(* PLC project Iec Unit Test, CODESYS CODESYS V3.5 SP16, author Toni Kucic *)
(* stored: creationDateTime 2021-05-10T20:20:27.8904239, version 0.1, modificationDateTime 2021-05-10T20:20:18.2154107, organization TK Automation *)
(* Library written in pure IEC 61131-3 Structured text that can be used for unit testing of any PLC POU. This library has arisen from the need of having a manufacturer and IDE independent unit test framework that is easily portable to other platform as the community requires. There are good unit frameworks existing for TwinCat, Codesys, B&R and many more platforms but none of them quite solve the extreme cases. *)

TYPE utTestCase : STRUCT
  id : UINT;  (* Identifier of the test *)
  desc : ARRAY[0..4] OF STRING(255);  (* Description of the test case *)
  state : utTestCaseStates;  (* State of the test *)
  msg : STRING(255);  (* Result of the test *)
END_STRUCT;
END_TYPE

(* values of utTestCaseStates: SETUP: Test case in setup mode, ready for execution; RUNNING: Test case running; PASSED: Test case passed; FAILED: Test case failed *)

{attribute 'qualified_only'}
{attribute 'strict'}
TYPE utTestCaseStates : (SETUP := 0, RUNNING := 1, PASSED := 2, FAILED := 3);
END_TYPE

TYPE utTestCaseSummary : STRUCT
  Id : UINT;  (* Id of the test object. Must be unique number *)
  Name : STRING(250);  (* Name of the test object *)
  TotalTests : UINT;  (* Total number of tests existing *)
  TestsPassed : UINT;  (* Number of tests passed *)
  TestsFailed : UINT;  (* Number of tests failed *)
  PassRate : REAL;  (* Pass rate % of the tests *)
  TestsRunning : BOOL;  (* One or more tests are running *)
  Error : utErrors := utErrors.NO_ERROR;  (* Error code if error occured *)
END_STRUCT;
END_TYPE

(* values of utErrors: NO_ERROR: No errors detected; NO_TEST_CASES_DEFINED: No test cases defined for this POU *)

{attribute 'qualified_only'}
{attribute 'strict'}
TYPE utErrors : (NO_ERROR := 0, NO_TEST_CASES_DEFINED := 100);
END_TYPE

FUNCTION assertFalse : BOOL
  VAR_INPUT
    condition : BOOL;  (* Variable to test *)
  END_VAR

            assertFalse := NOT condition;
RETURN;

          
END_FUNCTION

FUNCTION assertEqual_BOOL : BOOL
  VAR_INPUT
    act : BOOL;  (* Variable to test *)
    xp : BOOL;  (* Variable to test against *)
  END_VAR

            assertEqual_BOOL := act = xp;
RETURN;

          
END_FUNCTION

FUNCTION assertEqual_BYTE : BOOL
  VAR_INPUT
    act : BYTE;  (* Variable to test *)
    xp : BYTE;  (* Variable to test against *)
  END_VAR

            assertEqual_BYTE := act = xp;
RETURN;

          
END_FUNCTION

FUNCTION assertEqual_WORD : BOOL
  VAR_INPUT
    act : WORD;  (* Variable to test *)
    xp : WORD;  (* Variable to test against *)
  END_VAR

            assertEqual_WORD := act = xp;
RETURN;

          
END_FUNCTION

FUNCTION assertEqual_DWORD : BOOL
  VAR_INPUT
    act : DWORD;  (* Variable to test *)
    xp : DWORD;  (* Variable to test against *)
  END_VAR

            assertEqual_DWORD := act = xp;
RETURN;

          
END_FUNCTION

FUNCTION assertEqual_LWORD : BOOL
  VAR_INPUT
    act : LWORD;  (* Variable to test *)
    xp : LWORD;  (* Variable to test against *)
  END_VAR

            assertEqual_LWORD := act = xp;
RETURN;

          
END_FUNCTION

FUNCTION assertEqual_SINT : BOOL
  VAR_INPUT
    act : SINT;  (* Variable to test *)
    xp : SINT;  (* Variable to test against *)
  END_VAR

            assertEqual_SINT := act = xp;
RETURN;

          
END_FUNCTION

FUNCTION assertEqual_USINT : BOOL
  VAR_INPUT
    act : USINT;  (* Variable to test *)
    xp : USINT;  (* Variable to test against *)
  END_VAR

            assertEqual_USINT := act = xp;
RETURN;

          
END_FUNCTION

FUNCTION assertEqual_INT : BOOL
  VAR_INPUT
    act : INT;  (* Variable to test *)
    xp : INT;  (* Variable to test against *)
  END_VAR

            assertEqual_INT := act = xp;
RETURN;

          
END_FUNCTION

FUNCTION assertEqual_UINT : BOOL
  VAR_INPUT
    act : UINT;  (* Variable to test *)
    xp : UINT;  (* Variable to test against *)
  END_VAR

            assertEqual_UINT := act = xp;
RETURN;

          
END_FUNCTION

FUNCTION assertEqual_DINT : BOOL
  VAR_INPUT
    act : DINT;  (* Variable to test *)
    xp : DINT;  (* Variable to test against *)
  END_VAR

            assertEqual_DINT := act = xp;
RETURN;

          
END_FUNCTION

FUNCTION assertEqual_UDINT : BOOL
  VAR_INPUT
    act : UDINT;  (* Variable to test *)
    xp : UDINT;  (* Variable to test against *)
  END_VAR

            assertEqual_UDINT := act = xp;
RETURN;

          
END_FUNCTION

FUNCTION assertEqual_LINT : BOOL
  VAR_INPUT
    act : LINT;  (* Variable to test *)
    xp : LINT;  (* Variable to test against *)
  END_VAR

            assertEqual_LINT := act = xp;
RETURN;

          
END_FUNCTION

FUNCTION assertEqual_ULINT : BOOL
  VAR_INPUT
    act : ULINT;  (* Variable to test *)
    xp : ULINT;  (* Variable to test against *)
  END_VAR

            assertEqual_ULINT := act = xp;
RETURN;

          
END_FUNCTION

FUNCTION assertEqual_REAL : BOOL
  VAR_INPUT
    act : REAL;  (* Variable to test *)
    xp : REAL;  (* Variable to test against *)
  END_VAR

            assertEqual_REAL := act = xp;
RETURN;

          
END_FUNCTION

FUNCTION assertEqual_LREAL : BOOL
  VAR_INPUT
    act : LREAL;  (* Variable to test *)
    xp : LREAL;  (* Variable to test against *)
  END_VAR

            assertEqual_LREAL := act = xp;
RETURN;

          
END_FUNCTION

FUNCTION assertEqual_STRING : BOOL
  VAR_INPUT
    act : STRING;  (* Variable to test *)
    xp : STRING;  (* Variable to test against *)
  END_VAR

            assertEqual_STRING := act = xp;
RETURN;

          
END_FUNCTION

FUNCTION assertEqual_WSTRING : BOOL
  VAR_INPUT
    act : WSTRING;  (* Variable to test *)
    xp : WSTRING;  (* Variable to test against *)
  END_VAR

            assertEqual_WSTRING := act = xp;
RETURN;

          
END_FUNCTION

FUNCTION assertEqual_TIME : BOOL
  VAR_INPUT
    act : TIME;  (* Variable to test *)
    xp : TIME;  (* Variable to test against *)
  END_VAR

            assertEqual_TIME := act = xp;
RETURN;

          
END_FUNCTION

FUNCTION assertEqual_LTIME : BOOL
  VAR_INPUT
    act : LTIME;  (* Variable to test *)
    xp : LTIME;  (* Variable to test against *)
  END_VAR

            assertEqual_LTIME := act = xp;
RETURN;

          
END_FUNCTION

FUNCTION assertEqual_DATE : BOOL
  VAR_INPUT
    act : DATE;  (* Variable to test *)
    xp : DATE;  (* Variable to test against *)
  END_VAR

            assertEqual_DATE := act = xp;
RETURN;

          
END_FUNCTION

FUNCTION assertEqual_LDATE : BOOL
  VAR_INPUT
    act : LDATE;  (* Variable to test *)
    xp : LDATE;  (* Variable to test against *)
  END_VAR

            assertEqual_LDATE := act = xp;
RETURN;

          
END_FUNCTION

FUNCTION assertEqual_DATE_AND_TIME : BOOL
  VAR_INPUT
    act : DT;  (* Variable to test *)
    xp : DT;  (* Variable to test against *)
  END_VAR

            assertEqual_DATE_AND_TIME := act = xp;
RETURN;

          
END_FUNCTION

FUNCTION assertEqual_LDATE_AND_TIME : BOOL
  VAR_INPUT
    act : LDATE_AND_TIME;  (* Variable to test *)
    xp : LDATE_AND_TIME;  (* Variable to test against *)
  END_VAR

            assertEqual_LDATE_AND_TIME := act = xp;
RETURN;

          
END_FUNCTION

FUNCTION assertEqual_TIME_OF_DAY : BOOL
  VAR_INPUT
    act : TOD;  (* Variable to test *)
    xp : TOD;  (* Variable to test against *)
  END_VAR

            assertEqual_TIME_OF_DAY := act = xp;
RETURN;

          
END_FUNCTION

FUNCTION assertEqual_LTIME_OF_DAY : BOOL
  VAR_INPUT
    act : LTIME_OF_DAY;  (* Variable to test *)
    xp : LTIME_OF_DAY;  (* Variable to test against *)
  END_VAR

            assertEqual_LTIME_OF_DAY := act = xp;
RETURN;

          
END_FUNCTION

FUNCTION assertNotEqual_BOOL : BOOL
  VAR_INPUT
    act : BOOL;  (* Variable to test *)
    xp : BOOL;  (* Variable to test against *)
  END_VAR

            assertNotEqual_BOOL := act <> xp;
RETURN;

          
END_FUNCTION

FUNCTION assertNotEqual_BYTE : BOOL
  VAR_INPUT
    act : BYTE;  (* Variable to test *)
    xp : BYTE;  (* Variable to test against *)
  END_VAR

            assertNotEqual_BYTE := act <> xp;
RETURN;

          
END_FUNCTION

FUNCTION assertNotEqual_WORD : BOOL
  VAR_INPUT
    act : WORD;  (* Variable to test *)
    xp : WORD;  (* Variable to test against *)
  END_VAR

            assertNotEqual_WORD := act <> xp;
RETURN;

          
END_FUNCTION

FUNCTION assertNotEqual_DWORD : BOOL
  VAR_INPUT
    act : DWORD;  (* Variable to test *)
    xp : DWORD;  (* Variable to test against *)
  END_VAR

            assertNotEqual_DWORD := act <> xp;
RETURN;

          
END_FUNCTION

FUNCTION assertNotEqual_LWORD : BOOL
  VAR_INPUT
    act : LWORD;  (* Variable to test *)
    xp : LWORD;  (* Variable to test against *)
  END_VAR

            assertNotEqual_LWORD := act <> xp;
RETURN;

          
END_FUNCTION

FUNCTION assertNotEqual_SINT : BOOL
  VAR_INPUT
    act : SINT;  (* Variable to test *)
    xp : SINT;  (* Variable to test against *)
  END_VAR

            assertNotEqual_SINT := act <> xp;
RETURN;

          
END_FUNCTION

FUNCTION assertNotEqual_USINT : BOOL
  VAR_INPUT
    act : USINT;  (* Variable to test *)
    xp : USINT;  (* Variable to test against *)
  END_VAR

            assertNotEqual_USINT := act <> xp;
RETURN;

          
END_FUNCTION

FUNCTION assertNotEqual_INT : BOOL
  VAR_INPUT
    act : INT;  (* Variable to test *)
    xp : INT;  (* Variable to test against *)
  END_VAR

            assertNotEqual_INT := act <> xp;
RETURN;

          
END_FUNCTION

FUNCTION assertNotEqual_UINT : BOOL
  VAR_INPUT
    act : UINT;  (* Variable to test *)
    xp : UINT;  (* Variable to test against *)
  END_VAR

            assertNotEqual_UINT := act <> xp;
RETURN;

          
END_FUNCTION

FUNCTION assertNotEqual_DINT : BOOL
  VAR_INPUT
    act : DINT;  (* Variable to test *)
    xp : DINT;  (* Variable to test against *)
  END_VAR

            assertNotEqual_DINT := act <> xp;
RETURN;

          
END_FUNCTION

FUNCTION assertNotEqual_UDINT : BOOL
  VAR_INPUT
    act : UDINT;  (* Variable to test *)
    xp : UDINT;  (* Variable to test against *)
  END_VAR

            assertNotEqual_UDINT := act <> xp;
RETURN;

          
END_FUNCTION

FUNCTION assertNotEqual_LINT : BOOL
  VAR_INPUT
    act : LINT;  (* Variable to test *)
    xp : LINT;  (* Variable to test against *)
  END_VAR

            assertNotEqual_LINT := act <> xp;
RETURN;

          
END_FUNCTION

FUNCTION assertNotEqual_ULINT : BOOL
  VAR_INPUT
    act : ULINT;  (* Variable to test *)
    xp : ULINT;  (* Variable to test against *)
  END_VAR

            assertNotEqual_ULINT := act <> xp;
RETURN;

          
END_FUNCTION

FUNCTION assertNotEqual_REAL : BOOL
  VAR_INPUT
    act : REAL;  (* Variable to test *)
    xp : REAL;  (* Variable to test against *)
  END_VAR

            assertNotEqual_REAL := act <> xp;
RETURN;

          
END_FUNCTION

FUNCTION assertNotEqual_LREAL : BOOL
  VAR_INPUT
    act : LREAL;  (* Variable to test *)
    xp : LREAL;  (* Variable to test against *)
  END_VAR

            assertNotEqual_LREAL := act <> xp;
RETURN;

          
END_FUNCTION

FUNCTION assertNotEqual_STRING : BOOL
  VAR_INPUT
    act : STRING;  (* Variable to test *)
    xp : STRING;  (* Variable to test against *)
  END_VAR

            assertNotEqual_STRING := act <> xp;
RETURN;

          
END_FUNCTION

FUNCTION assertNotEqual_WSTRING : BOOL
  VAR_INPUT
    act : WSTRING;  (* Variable to test *)
    xp : WSTRING;  (* Variable to test against *)
  END_VAR

            assertNotEqual_WSTRING := act <> xp;
RETURN;

          
END_FUNCTION

FUNCTION assertNotEqual_TIME : BOOL
  VAR_INPUT
    act : TIME;  (* Variable to test *)
    xp : TIME;  (* Variable to test against *)
  END_VAR

            assertNotEqual_TIME := act <> xp;
RETURN;

          
END_FUNCTION

FUNCTION assertNotEqual_LTIME : BOOL
  VAR_INPUT
    act : LTIME;  (* Variable to test *)
    xp : LTIME;  (* Variable to test against *)
  END_VAR

            assertNotEqual_LTIME := act <> xp;
RETURN;

          
END_FUNCTION

FUNCTION assertNotEqual_DATE : BOOL
  VAR_INPUT
    act : DATE;  (* Variable to test *)
    xp : DATE;  (* Variable to test against *)
  END_VAR

            assertNotEqual_DATE := act <> xp;
RETURN;

          
END_FUNCTION

FUNCTION assertNotEqual_LDATE : BOOL
  VAR_INPUT
    act : LDATE;  (* Variable to test *)
    xp : LDATE;  (* Variable to test against *)
  END_VAR

            assertNotEqual_LDATE := act <> xp;
RETURN;

          
END_FUNCTION

FUNCTION assertNotEqual_DATE_AND_TIME : BOOL
  VAR_INPUT
    act : DT;  (* Variable to test *)
    xp : DT;  (* Variable to test against *)
  END_VAR

            assertNotEqual_DATE_AND_TIME := act <> xp;
RETURN;

          
END_FUNCTION

FUNCTION assertNotEqual_LDATE_AND_TIME : BOOL
  VAR_INPUT
    act : LDATE_AND_TIME;  (* Variable to test *)
    xp : LDATE_AND_TIME;  (* Variable to test against *)
  END_VAR

            assertNotEqual_LDATE_AND_TIME := act <> xp;
RETURN;

          
END_FUNCTION

FUNCTION assertNotEqual_TIME_OF_DAY : BOOL
  VAR_INPUT
    act : TOD;  (* Variable to test *)
    xp : TOD;  (* Variable to test against *)
  END_VAR

            assertNotEqual_TIME_OF_DAY := act <> xp;
RETURN;

          
END_FUNCTION

FUNCTION assertNotEqual_LTIME_OF_DAY : BOOL
  VAR_INPUT
    act : LTIME_OF_DAY;  (* Variable to test *)
    xp : LTIME_OF_DAY;  (* Variable to test against *)
  END_VAR

            assertNotEqual_LTIME_OF_DAY := act <> xp;
RETURN;

          
END_FUNCTION

FUNCTION assertGreater_BYTE : BOOL
  VAR_INPUT
    act : BYTE;  (* Variable to test *)
    xp : BYTE;  (* Variable to test against *)
  END_VAR

            assertGreater_BYTE := act > xp;
RETURN;

          
END_FUNCTION

FUNCTION assertGreater_WORD : BOOL
  VAR_INPUT
    act : WORD;  (* Variable to test *)
    xp : WORD;  (* Variable to test against *)
  END_VAR

            assertGreater_WORD := act > xp;
RETURN;

          
END_FUNCTION

FUNCTION assertGreater_DWORD : BOOL
  VAR_INPUT
    act : DWORD;  (* Variable to test *)
    xp : DWORD;  (* Variable to test against *)
  END_VAR

            assertGreater_DWORD := act > xp;
RETURN;

          
END_FUNCTION

FUNCTION assertGreater_LWORD : BOOL
  VAR_INPUT
    act : LWORD;  (* Variable to test *)
    xp : LWORD;  (* Variable to test against *)
  END_VAR

            assertGreater_LWORD := act > xp;
RETURN;

          
END_FUNCTION

FUNCTION assertGreater_SINT : BOOL
  VAR_INPUT
    act : SINT;  (* Variable to test *)
    xp : SINT;  (* Variable to test against *)
  END_VAR

            assertGreater_SINT := act > xp;
RETURN;

          
END_FUNCTION

FUNCTION assertGreater_USINT : BOOL
  VAR_INPUT
    act : USINT;  (* Variable to test *)
    xp : USINT;  (* Variable to test against *)
  END_VAR

            assertGreater_USINT := act > xp;
RETURN;

          
END_FUNCTION

FUNCTION assertGreater_INT : BOOL
  VAR_INPUT
    act : INT;  (* Variable to test *)
    xp : INT;  (* Variable to test against *)
  END_VAR

            assertGreater_INT := act > xp;
RETURN;

          
END_FUNCTION

FUNCTION assertGreater_UINT : BOOL
  VAR_INPUT
    act : UINT;  (* Variable to test *)
    xp : UINT;  (* Variable to test against *)
  END_VAR

            assertGreater_UINT := act > xp;
RETURN;

          
END_FUNCTION

FUNCTION assertGreater_DINT : BOOL
  VAR_INPUT
    act : DINT;  (* Variable to test *)
    xp : DINT;  (* Variable to test against *)
  END_VAR

            assertGreater_DINT := act > xp;
RETURN;

          
END_FUNCTION

FUNCTION assertGreater_UDINT : BOOL
  VAR_INPUT
    act : UDINT;  (* Variable to test *)
    xp : UDINT;  (* Variable to test against *)
  END_VAR

            assertGreater_UDINT := act > xp;
RETURN;

          
END_FUNCTION

FUNCTION assertGreater_LINT : BOOL
  VAR_INPUT
    act : LINT;  (* Variable to test *)
    xp : LINT;  (* Variable to test against *)
  END_VAR

            assertGreater_LINT := act > xp;
RETURN;

          
END_FUNCTION

FUNCTION assertGreater_ULINT : BOOL
  VAR_INPUT
    act : ULINT;  (* Variable to test *)
    xp : ULINT;  (* Variable to test against *)
  END_VAR

            assertGreater_ULINT := act > xp;
RETURN;

          
END_FUNCTION

FUNCTION assertGreater_REAL : BOOL
  VAR_INPUT
    act : REAL;  (* Variable to test *)
    xp : REAL;  (* Variable to test against *)
  END_VAR

            assertGreater_REAL := act > xp;
RETURN;

          
END_FUNCTION

FUNCTION assertGreater_LREAL : BOOL
  VAR_INPUT
    act : LREAL;  (* Variable to test *)
    xp : LREAL;  (* Variable to test against *)
  END_VAR

            assertGreater_LREAL := act > xp;
RETURN;

          
END_FUNCTION

FUNCTION assertGreater_TIME : BOOL
  VAR_INPUT
    act : TIME;  (* Variable to test *)
    xp : TIME;  (* Variable to test against *)
  END_VAR

            assertGreater_TIME := act > xp;
RETURN;

          
END_FUNCTION

FUNCTION assertGreater_LTIME : BOOL
  VAR_INPUT
    act : LTIME;  (* Variable to test *)
    xp : LTIME;  (* Variable to test against *)
  END_VAR

            assertGreater_LTIME := act > xp;
RETURN;

          
END_FUNCTION

FUNCTION assertGreater_DATE : BOOL
  VAR_INPUT
    act : DATE;  (* Variable to test *)
    xp : DATE;  (* Variable to test against *)
  END_VAR

            assertGreater_DATE := act > xp;
RETURN;

          
END_FUNCTION

FUNCTION assertGreater_LDATE : BOOL
  VAR_INPUT
    act : LDATE;  (* Variable to test *)
    xp : LDATE;  (* Variable to test against *)
  END_VAR

            assertGreater_LDATE := act > xp;
RETURN;

          
END_FUNCTION

FUNCTION assertGreater_DATE_AND_TIME : BOOL
  VAR_INPUT
    act : DT;  (* Variable to test *)
    xp : DT;  (* Variable to test against *)
  END_VAR

            assertGreater_DATE_AND_TIME := act > xp;
RETURN;

          
END_FUNCTION

FUNCTION assertGreater_LDATE_AND_TIME : BOOL
  VAR_INPUT
    act : LDATE_AND_TIME;  (* Variable to test *)
    xp : LDATE_AND_TIME;  (* Variable to test against *)
  END_VAR

            assertGreater_LDATE_AND_TIME := act > xp;
RETURN;

          
END_FUNCTION

FUNCTION assertGreater_TIME_OF_DAY : BOOL
  VAR_INPUT
    act : TOD;  (* Variable to test *)
    xp : TOD;  (* Variable to test against *)
  END_VAR

            assertGreater_TIME_OF_DAY := act > xp;
RETURN;

          
END_FUNCTION

FUNCTION assertGreater_LTIME_OF_DAY : BOOL
  VAR_INPUT
    act : LTIME_OF_DAY;  (* Variable to test *)
    xp : LTIME_OF_DAY;  (* Variable to test against *)
  END_VAR

            assertGreater_LTIME_OF_DAY := act > xp;
RETURN;

          
END_FUNCTION

FUNCTION assertGreaterEqual_BYTE : BOOL
  VAR_INPUT
    act : BYTE;  (* Variable to test *)
    xp : BYTE;  (* Variable to test against *)
  END_VAR

            assertGreaterEqual_BYTE := act >= xp;
RETURN;

          
END_FUNCTION

FUNCTION assertGreaterEqual_WORD : BOOL
  VAR_INPUT
    act : WORD;  (* Variable to test *)
    xp : WORD;  (* Variable to test against *)
  END_VAR

            assertGreaterEqual_WORD := act >= xp;
RETURN;

          
END_FUNCTION

FUNCTION assertGreaterEqual_DWORD : BOOL
  VAR_INPUT
    act : DWORD;  (* Variable to test *)
    xp : DWORD;  (* Variable to test against *)
  END_VAR

            assertGreaterEqual_DWORD := act >= xp;
RETURN;

          
END_FUNCTION

FUNCTION assertGreaterEqual_LWORD : BOOL
  VAR_INPUT
    act : LWORD;  (* Variable to test *)
    xp : LWORD;  (* Variable to test against *)
  END_VAR

            assertGreaterEqual_LWORD := act >= xp;
RETURN;

          
END_FUNCTION

FUNCTION assertGreaterEqual_SINT : BOOL
  VAR_INPUT
    act : SINT;  (* Variable to test *)
    xp : SINT;  (* Variable to test against *)
  END_VAR

            assertGreaterEqual_SINT := act >= xp;
RETURN;

          
END_FUNCTION

FUNCTION assertGreaterEqual_USINT : BOOL
  VAR_INPUT
    act : USINT;  (* Variable to test *)
    xp : USINT;  (* Variable to test against *)
  END_VAR

            assertGreaterEqual_USINT := act >= xp;
RETURN;

          
END_FUNCTION

FUNCTION assertGreaterEqual_INT : BOOL
  VAR_INPUT
    act : INT;  (* Variable to test *)
    xp : INT;  (* Variable to test against *)
  END_VAR

            assertGreaterEqual_INT := act >= xp;
RETURN;

          
END_FUNCTION

FUNCTION assertGreaterEqual_UINT : BOOL
  VAR_INPUT
    act : UINT;  (* Variable to test *)
    xp : UINT;  (* Variable to test against *)
  END_VAR

            assertGreaterEqual_UINT := act >= xp;
RETURN;

          
END_FUNCTION

FUNCTION assertGreaterEqual_DINT : BOOL
  VAR_INPUT
    act : DINT;  (* Variable to test *)
    xp : DINT;  (* Variable to test against *)
  END_VAR

            assertGreaterEqual_DINT := act >= xp;
RETURN;

          
END_FUNCTION

FUNCTION assertGreaterEqual_UDINT : BOOL
  VAR_INPUT
    act : UDINT;  (* Variable to test *)
    xp : UDINT;  (* Variable to test against *)
  END_VAR

            assertGreaterEqual_UDINT := act >= xp;
RETURN;

          
END_FUNCTION

FUNCTION assertGreaterEqual_LINT : BOOL
  VAR_INPUT
    act : LINT;  (* Variable to test *)
    xp : LINT;  (* Variable to test against *)
  END_VAR

            assertGreaterEqual_LINT := act >= xp;
RETURN;

          
END_FUNCTION

FUNCTION assertGreaterEqual_ULINT : BOOL
  VAR_INPUT
    act : ULINT;  (* Variable to test *)
    xp : ULINT;  (* Variable to test against *)
  END_VAR

            assertGreaterEqual_ULINT := act >= xp;
RETURN;

          
END_FUNCTION

FUNCTION assertGreaterEqual_REAL : BOOL
  VAR_INPUT
    act : REAL;  (* Variable to test *)
    xp : REAL;  (* Variable to test against *)
  END_VAR

            assertGreaterEqual_REAL := act >= xp;
RETURN;

          
END_FUNCTION

FUNCTION assertGreaterEqual_LREAL : BOOL
  VAR_INPUT
    act : LREAL;  (* Variable to test *)
    xp : LREAL;  (* Variable to test against *)
  END_VAR

            assertGreaterEqual_LREAL := act >= xp;
RETURN;

          
END_FUNCTION

FUNCTION assertGreaterEqual_TIME : BOOL
  VAR_INPUT
    act : TIME;  (* Variable to test *)
    xp : TIME;  (* Variable to test against *)
  END_VAR

            assertGreaterEqual_TIME := act >= xp;
RETURN;

          
END_FUNCTION

FUNCTION assertGreaterEqual_LTIME : BOOL
  VAR_INPUT
    act : LTIME;  (* Variable to test *)
    xp : LTIME;  (* Variable to test against *)
  END_VAR

            assertGreaterEqual_LTIME := act >= xp;
RETURN;

          
END_FUNCTION

FUNCTION assertGreaterEqual_DATE : BOOL
  VAR_INPUT
    act : DATE;  (* Variable to test *)
    xp : DATE;  (* Variable to test against *)
  END_VAR

            assertGreaterEqual_DATE := act >= xp;
RETURN;

          
END_FUNCTION

FUNCTION assertGreaterEqual_LDATE : BOOL
  VAR_INPUT
    act : LDATE;  (* Variable to test *)
    xp : LDATE;  (* Variable to test against *)
  END_VAR

            assertGreaterEqual_LDATE := act >= xp;
RETURN;

          
END_FUNCTION

FUNCTION assertGreaterEqual_DATE_AND_TIME : BOOL
  VAR_INPUT
    act : DT;  (* Variable to test *)
    xp : DT;  (* Variable to test against *)
  END_VAR

            assertGreaterEqual_DATE_AND_TIME := act >= xp;
RETURN;

          
END_FUNCTION

FUNCTION assertGreaterEqual_LDATE_AND_TIME : BOOL
  VAR_INPUT
    act : LDATE_AND_TIME;  (* Variable to test *)
    xp : LDATE_AND_TIME;  (* Variable to test against *)
  END_VAR

            assertGreaterEqual_LDATE_AND_TIME := act >= xp;
RETURN;

          
END_FUNCTION

FUNCTION assertGreaterEqual_TIME_OF_DAY : BOOL
  VAR_INPUT
    act : TOD;  (* Variable to test *)
    xp : TOD;  (* Variable to test against *)
  END_VAR

            assertGreaterEqual_TIME_OF_DAY := act >= xp;
RETURN;

          
END_FUNCTION

FUNCTION assertGreaterEqual_LTIME_OF_DAY : BOOL
  VAR_INPUT
    act : LTIME_OF_DAY;  (* Variable to test *)
    xp : LTIME_OF_DAY;  (* Variable to test against *)
  END_VAR

            assertGreaterEqual_LTIME_OF_DAY := act >= xp;
RETURN;

          
END_FUNCTION

FUNCTION assertLess_BYTE : BOOL
  VAR_INPUT
    act : BYTE;  (* Variable to test *)
    xp : BYTE;  (* Variable to test against *)
  END_VAR

            assertLess_BYTE := act < xp;
RETURN;

          
END_FUNCTION

FUNCTION assertLess_WORD : BOOL
  VAR_INPUT
    act : WORD;  (* Variable to test *)
    xp : WORD;  (* Variable to test against *)
  END_VAR

            assertLess_WORD := act < xp;
RETURN;

          
END_FUNCTION

FUNCTION assertLess_DWORD : BOOL
  VAR_INPUT
    act : DWORD;  (* Variable to test *)
    xp : DWORD;  (* Variable to test against *)
  END_VAR

            assertLess_DWORD := act < xp;
RETURN;

          
END_FUNCTION

FUNCTION assertLess_LWORD : BOOL
  VAR_INPUT
    act : LWORD;  (* Variable to test *)
    xp : LWORD;  (* Variable to test against *)
  END_VAR

            assertLess_LWORD := act < xp;
RETURN;

          
END_FUNCTION

FUNCTION assertLess_SINT : BOOL
  VAR_INPUT
    act : SINT;  (* Variable to test *)
    xp : SINT;  (* Variable to test against *)
  END_VAR

            assertLess_SINT := act < xp;
RETURN;

          
END_FUNCTION

FUNCTION assertLess_USINT : BOOL
  VAR_INPUT
    act : USINT;  (* Variable to test *)
    xp : USINT;  (* Variable to test against *)
  END_VAR

            assertLess_USINT := act < xp;
RETURN;

          
END_FUNCTION

FUNCTION assertLess_INT : BOOL
  VAR_INPUT
    act : INT;  (* Variable to test *)
    xp : INT;  (* Variable to test against *)
  END_VAR

            assertLess_INT := act < xp;
RETURN;

          
END_FUNCTION

FUNCTION assertLess_UINT : BOOL
  VAR_INPUT
    act : UINT;  (* Variable to test *)
    xp : UINT;  (* Variable to test against *)
  END_VAR

            assertLess_UINT := act < xp;
RETURN;

          
END_FUNCTION

FUNCTION assertLess_DINT : BOOL
  VAR_INPUT
    act : DINT;  (* Variable to test *)
    xp : DINT;  (* Variable to test against *)
  END_VAR

            assertLess_DINT := act < xp;
RETURN;

          
END_FUNCTION

FUNCTION assertLess_UDINT : BOOL
  VAR_INPUT
    act : UDINT;  (* Variable to test *)
    xp : UDINT;  (* Variable to test against *)
  END_VAR

            assertLess_UDINT := act < xp;
RETURN;

          
END_FUNCTION

FUNCTION assertLess_LINT : BOOL
  VAR_INPUT
    act : LINT;  (* Variable to test *)
    xp : LINT;  (* Variable to test against *)
  END_VAR

            assertLess_LINT := act < xp;
RETURN;

          
END_FUNCTION

FUNCTION assertLess_ULINT : BOOL
  VAR_INPUT
    act : ULINT;  (* Variable to test *)
    xp : ULINT;  (* Variable to test against *)
  END_VAR

            assertLess_ULINT := act < xp;
RETURN;

          
END_FUNCTION

FUNCTION assertLess_REAL : BOOL
  VAR_INPUT
    act : REAL;  (* Variable to test *)
    xp : REAL;  (* Variable to test against *)
  END_VAR

            assertLess_REAL := act < xp;
RETURN;

          
END_FUNCTION

FUNCTION assertLess_LREAL : BOOL
  VAR_INPUT
    act : LREAL;  (* Variable to test *)
    xp : LREAL;  (* Variable to test against *)
  END_VAR

            assertLess_LREAL := act < xp;
RETURN;

          
END_FUNCTION

FUNCTION assertLess_TIME : BOOL
  VAR_INPUT
    act : TIME;  (* Variable to test *)
    xp : TIME;  (* Variable to test against *)
  END_VAR

            assertLess_TIME := act < xp;
RETURN;

          
END_FUNCTION

FUNCTION assertLess_LTIME : BOOL
  VAR_INPUT
    act : LTIME;  (* Variable to test *)
    xp : LTIME;  (* Variable to test against *)
  END_VAR

            assertLess_LTIME := act < xp;
RETURN;

          
END_FUNCTION

FUNCTION assertLess_DATE : BOOL
  VAR_INPUT
    act : DATE;  (* Variable to test *)
    xp : DATE;  (* Variable to test against *)
  END_VAR

            assertLess_DATE := act < xp;
RETURN;

          
END_FUNCTION

FUNCTION assertLess_LDATE : BOOL
  VAR_INPUT
    act : LDATE;  (* Variable to test *)
    xp : LDATE;  (* Variable to test against *)
  END_VAR

            assertLess_LDATE := act < xp;
RETURN;

          
END_FUNCTION

FUNCTION assertLess_DATE_AND_TIME : BOOL
  VAR_INPUT
    act : DT;  (* Variable to test *)
    xp : DT;  (* Variable to test against *)
  END_VAR

            assertLess_DATE_AND_TIME := act < xp;
RETURN;

          
END_FUNCTION

FUNCTION assertLess_LDATE_AND_TIME : BOOL
  VAR_INPUT
    act : LDATE_AND_TIME;  (* Variable to test *)
    xp : LDATE_AND_TIME;  (* Variable to test against *)
  END_VAR

            assertLess_LDATE_AND_TIME := act < xp;
RETURN;

          
END_FUNCTION

FUNCTION assertLess_TIME_OF_DAY : BOOL
  VAR_INPUT
    act : TOD;  (* Variable to test *)
    xp : TOD;  (* Variable to test against *)
  END_VAR

            assertLess_TIME_OF_DAY := act < xp;
RETURN;

          
END_FUNCTION

FUNCTION assertLess_LTIME_OF_DAY : BOOL
  VAR_INPUT
    act : LTIME_OF_DAY;  (* Variable to test *)
    xp : LTIME_OF_DAY;  (* Variable to test against *)
  END_VAR

            assertLess_LTIME_OF_DAY := act < xp;
RETURN;

          
END_FUNCTION

FUNCTION assertLessEqual_BYTE : BOOL
  VAR_INPUT
    act : BYTE;  (* Variable to test *)
    xp : BYTE;  (* Variable to test against *)
  END_VAR

            assertLessEqual_BYTE := act <= xp;
RETURN;

          
END_FUNCTION

FUNCTION assertLessEqual_WORD : BOOL
  VAR_INPUT
    act : WORD;  (* Variable to test *)
    xp : WORD;  (* Variable to test against *)
  END_VAR

            assertLessEqual_WORD := act <= xp;
RETURN;

          
END_FUNCTION

FUNCTION assertLessEqual_DWORD : BOOL
  VAR_INPUT
    act : DWORD;  (* Variable to test *)
    xp : DWORD;  (* Variable to test against *)
  END_VAR

            assertLessEqual_DWORD := act <= xp;
RETURN;

          
END_FUNCTION

FUNCTION assertLessEqual_LWORD : BOOL
  VAR_INPUT
    act : LWORD;  (* Variable to test *)
    xp : LWORD;  (* Variable to test against *)
  END_VAR

            assertLessEqual_LWORD := act <= xp;
RETURN;

          
END_FUNCTION

FUNCTION assertLessEqual_SINT : BOOL
  VAR_INPUT
    act : SINT;  (* Variable to test *)
    xp : SINT;  (* Variable to test against *)
  END_VAR

            assertLessEqual_SINT := act <= xp;
RETURN;

          
END_FUNCTION

FUNCTION assertLessEqual_USINT : BOOL
  VAR_INPUT
    act : USINT;  (* Variable to test *)
    xp : USINT;  (* Variable to test against *)
  END_VAR

            assertLessEqual_USINT := act <= xp;
RETURN;

          
END_FUNCTION

FUNCTION assertLessEqual_INT : BOOL
  VAR_INPUT
    act : INT;  (* Variable to test *)
    xp : INT;  (* Variable to test against *)
  END_VAR

            assertLessEqual_INT := act <= xp;
RETURN;

          
END_FUNCTION

FUNCTION assertLessEqual_UINT : BOOL
  VAR_INPUT
    act : UINT;  (* Variable to test *)
    xp : UINT;  (* Variable to test against *)
  END_VAR

            assertLessEqual_UINT := act <= xp;
RETURN;

          
END_FUNCTION

FUNCTION assertLessEqual_DINT : BOOL
  VAR_INPUT
    act : DINT;  (* Variable to test *)
    xp : DINT;  (* Variable to test against *)
  END_VAR

            assertLessEqual_DINT := act <= xp;
RETURN;

          
END_FUNCTION

FUNCTION assertLessEqual_UDINT : BOOL
  VAR_INPUT
    act : UDINT;  (* Variable to test *)
    xp : UDINT;  (* Variable to test against *)
  END_VAR

            assertLessEqual_UDINT := act <= xp;
RETURN;

          
END_FUNCTION

FUNCTION assertLessEqual_LINT : BOOL
  VAR_INPUT
    act : LINT;  (* Variable to test *)
    xp : LINT;  (* Variable to test against *)
  END_VAR

            assertLessEqual_LINT := act <= xp;
RETURN;

          
END_FUNCTION

FUNCTION assertLessEqual_ULINT : BOOL
  VAR_INPUT
    act : ULINT;  (* Variable to test *)
    xp : ULINT;  (* Variable to test against *)
  END_VAR

            assertLessEqual_ULINT := act <= xp;
RETURN;

          
END_FUNCTION

FUNCTION assertLessEqual_REAL : BOOL
  VAR_INPUT
    act : REAL;  (* Variable to test *)
    xp : REAL;  (* Variable to test against *)
  END_VAR

            assertLessEqual_REAL := act <= xp;
RETURN;

          
END_FUNCTION

FUNCTION assertLessEqual_LREAL : BOOL
  VAR_INPUT
    act : LREAL;  (* Variable to test *)
    xp : LREAL;  (* Variable to test against *)
  END_VAR

            assertLessEqual_LREAL := act <= xp;
RETURN;

          
END_FUNCTION

FUNCTION assertLessEqual_TIME : BOOL
  VAR_INPUT
    act : TIME;  (* Variable to test *)
    xp : TIME;  (* Variable to test against *)
  END_VAR

            assertLessEqual_TIME := act <= xp;
RETURN;

          
END_FUNCTION

FUNCTION assertLessEqual_LTIME : BOOL
  VAR_INPUT
    act : LTIME;  (* Variable to test *)
    xp : LTIME;  (* Variable to test against *)
  END_VAR

            assertLessEqual_LTIME := act <= xp;
RETURN;

          
END_FUNCTION

FUNCTION assertLessEqual_DATE : BOOL
  VAR_INPUT
    act : DATE;  (* Variable to test *)
    xp : DATE;  (* Variable to test against *)
  END_VAR

            assertLessEqual_DATE := act <= xp;
RETURN;

          
END_FUNCTION

FUNCTION assertLessEqual_LDATE : BOOL
  VAR_INPUT
    act : LDATE;  (* Variable to test *)
    xp : LDATE;  (* Variable to test against *)
  END_VAR

            assertLessEqual_LDATE := act <= xp;
RETURN;

          
END_FUNCTION

FUNCTION assertLessEqual_DATE_AND_TIME : BOOL
  VAR_INPUT
    act : DT;  (* Variable to test *)
    xp : DT;  (* Variable to test against *)
  END_VAR

            assertLessEqual_DATE_AND_TIME := act <= xp;
RETURN;

          
END_FUNCTION

FUNCTION assertLessEqual_LDATE_AND_TIME : BOOL
  VAR_INPUT
    act : LDATE_AND_TIME;  (* Variable to test *)
    xp : LDATE_AND_TIME;  (* Variable to test against *)
  END_VAR

            assertLessEqual_LDATE_AND_TIME := act <= xp;
RETURN;

          
END_FUNCTION

FUNCTION assertLessEqual_TIME_OF_DAY : BOOL
  VAR_INPUT
    act : TOD;  (* Variable to test *)
    xp : TOD;  (* Variable to test against *)
  END_VAR

            assertLessEqual_TIME_OF_DAY := act <= xp;
RETURN;

          
END_FUNCTION

FUNCTION assertLessEqual_LTIME_OF_DAY : BOOL
  VAR_INPUT
    act : LTIME_OF_DAY;  (* Variable to test *)
    xp : LTIME_OF_DAY;  (* Variable to test against *)
  END_VAR

            assertLessEqual_LTIME_OF_DAY := act <= xp;
RETURN;

          
END_FUNCTION

FUNCTION assertArrayEqual_BOOL : BOOL
  VAR_INPUT
    act : POINTER TO ARRAY[0..32000] OF BOOL;  (* Variable to test *)
    xp : POINTER TO ARRAY[0..32000] OF BOOL;  (* Variable to test against *)
    size : UINT;  (* Size of the array (ADR(act)) *)
  END_VAR
  VAR
    i : UINT;  (* Iterator variable *)
    vStop : UINT;  (* Size of the array / End of iteration *)
    pt1 : POINTER TO BOOL;  (* Pointer to the element of the array act *)
    pt2 : POINTER TO BOOL;  (* Pointer to the element of the array xp *)
  END_VAR

            vStop := (size / SIZEOF(act^[0])) - 1;

FOR i:=0 TO vStop DO
	pt1 := ADR(act^[i]);
	pt2 := ADR(xp^[i]);
	IF pt1^ <> pt2^ THEN
		assertArrayEqual_BOOL := FALSE;
		RETURN;
	END_IF
END_FOR
(*If we reach here, all elements are equal*)
assertArrayEqual_BOOL := TRUE;
RETURN;

          
END_FUNCTION

FUNCTION assertArrayEqual_BYTE : BOOL
  VAR_INPUT
    act : POINTER TO ARRAY[0..32000] OF BYTE;  (* Variable to test *)
    xp : POINTER TO ARRAY[0..32000] OF BYTE;  (* Variable to test against *)
    size : UINT;  (* Size of the array (ADR(act)) *)
  END_VAR
  VAR
    i : UINT;  (* Iterator variable *)
    vStop : UINT;  (* Size of the array / End of iteration *)
    pt1 : POINTER TO BYTE;  (* Pointer to the element of the array act *)
    pt2 : POINTER TO BYTE;  (* Pointer to the element of the array xp *)
  END_VAR

            vStop := (size / SIZEOF(act^[0])) - 1;

FOR i:=0 TO vStop DO
	pt1 := ADR(act^[i]);
	pt2 := ADR(xp^[i]);
	IF pt1^ <> pt2^ THEN
		assertArrayEqual_BYTE := FALSE;
		RETURN;
	END_IF
END_FOR
(*If we reach here, all elements are equal*)
assertArrayEqual_BYTE := TRUE;
RETURN;

          
END_FUNCTION

FUNCTION assertArrayEqual_WORD : BOOL
  VAR_INPUT
    act : POINTER TO ARRAY[0..32000] OF WORD;  (* Variable to test *)
    xp : POINTER TO ARRAY[0..32000] OF WORD;  (* Variable to test against *)
    size : UINT;  (* Size of the array (ADR(act)) *)
  END_VAR
  VAR
    i : UINT;  (* Iterator variable *)
    vStop : UINT;  (* Size of the array / End of iteration *)
    pt1 : POINTER TO WORD;  (* Pointer to the element of the array act *)
    pt2 : POINTER TO WORD;  (* Pointer to the element of the array xp *)
  END_VAR

            vStop := (size / SIZEOF(act^[0])) - 1;

FOR i:=0 TO vStop DO
	pt1 := ADR(act^[i]);
	pt2 := ADR(xp^[i]);
	IF pt1^ <> pt2^ THEN
		assertArrayEqual_WORD := FALSE;
		RETURN;
	END_IF
END_FOR
(*If we reach here, all elements are equal*)
assertArrayEqual_WORD := TRUE;
RETURN;

          
END_FUNCTION

(* Returns TRUE if act == xp. *)
FUNCTION assertArrayEqual_DWORD : BOOL
  VAR_INPUT
    act : POINTER TO ARRAY[0..32000] OF DWORD;  (* Variable to test *)
    xp : POINTER TO ARRAY[0..32000] OF DWORD;  (* Variable to test against *)
    size : UINT;  (* Size of the array (ADR(act)) *)
  END_VAR
  VAR
    i : UINT;  (* Iterator variable *)
    vStop : UINT;  (* Size of the array / End of iteration *)
    pt1 : POINTER TO DWORD;  (* Pointer to the element of the array act *)
    pt2 : POINTER TO DWORD;  (* Pointer to the element of the array xp *)
  END_VAR

            vStop := (size / SIZEOF(act^[0])) - 1;

FOR i:=0 TO vStop DO
	pt1 := ADR(act^[i]);
	pt2 := ADR(xp^[i]);
	IF pt1^ <> pt2^ THEN
		assertArrayEqual_DWORD := FALSE;
		RETURN;
	END_IF
END_FOR
(*If we reach here, all elements are equal*)
assertArrayEqual_DWORD := TRUE;
RETURN;

          
END_FUNCTION

FUNCTION assertArrayEqual_LWORD : BOOL
  VAR_INPUT
    act : POINTER TO ARRAY[0..32000] OF LWORD;  (* Variable to test *)
    xp : POINTER TO ARRAY[0..32000] OF LWORD;  (* Variable to test against *)
    size : UINT;  (* Size of the array (ADR(act)) *)
  END_VAR
  VAR
    i : UINT;  (* Iterator variable *)
    vStop : UINT;  (* Size of the array / End of iteration *)
    pt1 : POINTER TO LWORD;  (* Pointer to the element of the array act *)
    pt2 : POINTER TO LWORD;  (* Pointer to the element of the array xp *)
  END_VAR

            vStop := (size / SIZEOF(act^[0])) - 1;

FOR i:=0 TO vStop DO
	pt1 := ADR(act^[i]);
	pt2 := ADR(xp^[i]);
	IF pt1^ <> pt2^ THEN
		assertArrayEqual_LWORD := FALSE;
		RETURN;
	END_IF
END_FOR
(*If we reach here, all elements are equal*)
assertArrayEqual_LWORD := TRUE;
RETURN;

          
END_FUNCTION

FUNCTION assertArrayEqual_SINT : BOOL
  VAR_INPUT
    act : POINTER TO ARRAY[0..32000] OF SINT;  (* Variable to test *)
    xp : POINTER TO ARRAY[0..32000] OF SINT;  (* Variable to test against *)
    size : UINT;  (* Size of the array (ADR(act)) *)
  END_VAR
  VAR
    i : UINT;  (* Iterator variable *)
    vStop : UINT;  (* Size of the array / End of iteration *)
    pt1 : POINTER TO SINT;  (* Pointer to the element of the array act *)
    pt2 : POINTER TO SINT;  (* Pointer to the element of the array xp *)
  END_VAR

            vStop := (size / SIZEOF(act^[0])) - 1;

FOR i:=0 TO vStop DO
	pt1 := ADR(act^[i]);
	pt2 := ADR(xp^[i]);
	IF pt1^ <> pt2^ THEN
		assertArrayEqual_SINT := FALSE;
		RETURN;
	END_IF
END_FOR
(*If we reach here, all elements are equal*)
assertArrayEqual_SINT := TRUE;
RETURN;

          
END_FUNCTION

FUNCTION assertArrayEqual_USINT : BOOL
  VAR_INPUT
    act : POINTER TO ARRAY[0..32000] OF USINT;  (* Variable to test *)
    xp : POINTER TO ARRAY[0..32000] OF USINT;  (* Variable to test against *)
    size : UINT;  (* Size of the array (ADR(act)) *)
  END_VAR
  VAR
    i : UINT;  (* Iterator variable *)
    vStop : UINT;  (* Size of the array / End of iteration *)
    pt1 : POINTER TO USINT;  (* Pointer to the element of the array act *)
    pt2 : POINTER TO USINT;  (* Pointer to the element of the array xp *)
  END_VAR

            vStop := (size / SIZEOF(act^[0])) - 1;

FOR i:=0 TO vStop DO
	pt1 := ADR(act^[i]);
	pt2 := ADR(xp^[i]);
	IF pt1^ <> pt2^ THEN
		assertArrayEqual_USINT := FALSE;
		RETURN;
	END_IF
END_FOR
(*If we reach here, all elements are equal*)
assertArrayEqual_USINT := TRUE;
RETURN;

          
END_FUNCTION

FUNCTION assertArrayEqual_INT : BOOL
  VAR_INPUT
    act : POINTER TO ARRAY[0..32000] OF INT;  (* Variable to test *)
    xp : POINTER TO ARRAY[0..32000] OF INT;  (* Variable to test against *)
    size : UINT;  (* Size of the array (ADR(act)) *)
  END_VAR
  VAR
    i : UINT;  (* Iterator variable *)
    vStop : UINT;  (* Size of the array / End of iteration *)
    pt1 : POINTER TO INT;  (* Pointer to the element of the array act *)
    pt2 : POINTER TO INT;  (* Pointer to the element of the array xp *)
  END_VAR

            vStop := (size / SIZEOF(act^[0])) - 1;

FOR i:=0 TO vStop DO
	pt1 := ADR(act^[i]);
	pt2 := ADR(xp^[i]);
	IF pt1^ <> pt2^ THEN
		assertArrayEqual_INT := FALSE;
		RETURN;
	END_IF
END_FOR
(*If we reach here, all elements are equal*)
assertArrayEqual_INT := TRUE;
RETURN;

          
END_FUNCTION

FUNCTION assertArrayEqual_UINT : BOOL
  VAR_INPUT
    act : POINTER TO ARRAY[0..32000] OF UINT;  (* Variable to test *)
    xp : POINTER TO ARRAY[0..32000] OF UINT;  (* Variable to test against *)
    size : UINT;  (* Size of the array (ADR(act)) *)
  END_VAR
  VAR
    i : UINT;  (* Iterator variable *)
    vStop : UINT;  (* Size of the array / End of iteration *)
    pt1 : POINTER TO UINT;  (* Pointer to the element of the array act *)
    pt2 : POINTER TO UINT;  (* Pointer to the element of the array xp *)
  END_VAR

            vStop := (size / SIZEOF(act^[0])) - 1;

FOR i:=0 TO vStop DO
	pt1 := ADR(act^[i]);
	pt2 := ADR(xp^[i]);
	IF pt1^ <> pt2^ THEN
		assertArrayEqual_UINT := FALSE;
		RETURN;
	END_IF
END_FOR
(*If we reach here, all elements are equal*)
assertArrayEqual_UINT := TRUE;
RETURN;

          
END_FUNCTION

FUNCTION assertArrayEqual_DINT : BOOL
  VAR_INPUT
    act : POINTER TO ARRAY[0..32000] OF DINT;  (* Variable to test *)
    xp : POINTER TO ARRAY[0..32000] OF DINT;  (* Variable to test against *)
    size : UINT;  (* Size of the array (ADR(act)) *)
  END_VAR
  VAR
    i : UINT;  (* Iterator variable *)
    vStop : UINT;  (* Size of the array / End of iteration *)
    pt1 : POINTER TO DINT;  (* Pointer to the element of the array act *)
    pt2 : POINTER TO DINT;  (* Pointer to the element of the array xp *)
  END_VAR

            vStop := (size / SIZEOF(act^[0])) - 1;

FOR i:=0 TO vStop DO
	pt1 := ADR(act^[i]);
	pt2 := ADR(xp^[i]);
	IF pt1^ <> pt2^ THEN
		assertArrayEqual_DINT := FALSE;
		RETURN;
	END_IF
END_FOR
(*If we reach here, all elements are equal*)
assertArrayEqual_DINT := TRUE;
RETURN;

          
END_FUNCTION

FUNCTION assertArrayEqual_UDINT : BOOL
  VAR_INPUT
    act : POINTER TO ARRAY[0..32000] OF UDINT;  (* Variable to test *)
    xp : POINTER TO ARRAY[0..32000] OF UDINT;  (* Variable to test against *)
    size : UINT;  (* Size of the array (ADR(act)) *)
  END_VAR
  VAR
    i : UINT;  (* Iterator variable *)
    vStop : UINT;  (* Size of the array / End of iteration *)
    pt1 : POINTER TO UDINT;  (* Pointer to the element of the array act *)
    pt2 : POINTER TO UDINT;  (* Pointer to the element of the array xp *)
  END_VAR

            vStop := (size / SIZEOF(act^[0])) - 1;

FOR i:=0 TO vStop DO
	pt1 := ADR(act^[i]);
	pt2 := ADR(xp^[i]);
	IF pt1^ <> pt2^ THEN
		assertArrayEqual_UDINT := FALSE;
		RETURN;
	END_IF
END_FOR
(*If we reach here, all elements are equal*)
assertArrayEqual_UDINT := TRUE;
RETURN;

          
END_FUNCTION

FUNCTION assertArrayEqual_LINT : BOOL
  VAR_INPUT
    act : POINTER TO ARRAY[0..32000] OF LINT;  (* Variable to test *)
    xp : POINTER TO ARRAY[0..32000] OF LINT;  (* Variable to test against *)
    size : UINT;  (* Size of the array (ADR(act)) *)
  END_VAR
  VAR
    i : UINT;  (* Iterator variable *)
    vStop : UINT;  (* Size of the array / End of iteration *)
    pt1 : POINTER TO LINT;  (* Pointer to the element of the array act *)
    pt2 : POINTER TO LINT;  (* Pointer to the element of the array xp *)
  END_VAR

            vStop := (size / SIZEOF(act^[0])) - 1;

FOR i:=0 TO vStop DO
	pt1 := ADR(act^[i]);
	pt2 := ADR(xp^[i]);
	IF pt1^ <> pt2^ THEN
		assertArrayEqual_LINT := FALSE;
		RETURN;
	END_IF
END_FOR
(*If we reach here, all elements are equal*)
assertArrayEqual_LINT := TRUE;
RETURN;

          
END_FUNCTION

FUNCTION assertArrayEqual_ULINT : BOOL
  VAR_INPUT
    act : POINTER TO ARRAY[0..32000] OF ULINT;  (* Variable to test *)
    xp : POINTER TO ARRAY[0..32000] OF ULINT;  (* Variable to test against *)
    size : UINT;  (* Size of the array (ADR(act)) *)
  END_VAR
  VAR
    i : UINT;  (* Iterator variable *)
    vStop : UINT;  (* Size of the array / End of iteration *)
    pt1 : POINTER TO ULINT;  (* Pointer to the element of the array act *)
    pt2 : POINTER TO ULINT;  (* Pointer to the element of the array xp *)
  END_VAR

            vStop := (size / SIZEOF(act^[0])) - 1;

FOR i:=0 TO vStop DO
	pt1 := ADR(act^[i]);
	pt2 := ADR(xp^[i]);
	IF pt1^ <> pt2^ THEN
		assertArrayEqual_ULINT := FALSE;
		RETURN;
	END_IF
END_FOR
(*If we reach here, all elements are equal*)
assertArrayEqual_ULINT := TRUE;
RETURN;

          
END_FUNCTION

FUNCTION assertArrayEqual_REAL : BOOL
  VAR_INPUT
    act : POINTER TO ARRAY[0..32000] OF REAL;  (* Variable to test *)
    xp : POINTER TO ARRAY[0..32000] OF REAL;  (* Variable to test against *)
    size : UINT;  (* Size of the array (ADR(act)) *)
  END_VAR
  VAR
    i : UINT;  (* Iterator variable *)
    vStop : UINT;  (* Size of the array / End of iteration *)
    pt1 : POINTER TO REAL;  (* Pointer to the element of the array act *)
    pt2 : POINTER TO REAL;  (* Pointer to the element of the array xp *)
  END_VAR

            vStop := (size / SIZEOF(act^[0])) - 1;

FOR i:=0 TO vStop DO
	pt1 := ADR(act^[i]);
	pt2 := ADR(xp^[i]);
	IF pt1^ <> pt2^ THEN
		assertArrayEqual_REAL := FALSE;
		RETURN;
	END_IF
END_FOR
(*If we reach here, all elements are equal*)
assertArrayEqual_REAL := TRUE;
RETURN;

          
END_FUNCTION

FUNCTION assertArrayEqual_LREAL : BOOL
  VAR_INPUT
    act : POINTER TO ARRAY[0..32000] OF LREAL;  (* Variable to test *)
    xp : POINTER TO ARRAY[0..32000] OF LREAL;  (* Variable to test against *)
    size : UINT;  (* Size of the array (ADR(act)) *)
  END_VAR
  VAR
    i : UINT;  (* Iterator variable *)
    vStop : UINT;  (* Size of the array / End of iteration *)
    pt1 : POINTER TO LREAL;  (* Pointer to the element of the array act *)
    pt2 : POINTER TO LREAL;  (* Pointer to the element of the array xp *)
  END_VAR

            vStop := (size / SIZEOF(act^[0])) - 1;

FOR i:=0 TO vStop DO
	pt1 := ADR(act^[i]);
	pt2 := ADR(xp^[i]);
	IF pt1^ <> pt2^ THEN
		assertArrayEqual_LREAL := FALSE;
		RETURN;
	END_IF
END_FOR
(*If we reach here, all elements are equal*)
assertArrayEqual_LREAL := TRUE;
RETURN;

          
END_FUNCTION

FUNCTION assertArrayEqual_STRING : BOOL
  VAR_INPUT
    act : POINTER TO ARRAY[0..32000] OF STRING;  (* Variable to test *)
    xp : POINTER TO ARRAY[0..32000] OF STRING;  (* Variable to test against *)
    size : UINT;  (* Size of the array (ADR(act)) *)
  END_VAR
  VAR
    i : UINT;  (* Iterator variable *)
    vStop : UINT;  (* Size of the array / End of iteration *)
    pt1 : POINTER TO STRING;  (* Pointer to the element of the array act *)
    pt2 : POINTER TO STRING;  (* Pointer to the element of the array xp *)
  END_VAR

            vStop := (size / SIZEOF(act^[0])) - 1;

FOR i:=0 TO vStop DO
	pt1 := ADR(act^[i]);
	pt2 := ADR(xp^[i]);
	IF pt1^ <> pt2^ THEN
		assertArrayEqual_STRING := FALSE;
		RETURN;
	END_IF
END_FOR
(*If we reach here, all elements are equal*)
assertArrayEqual_STRING := TRUE;
RETURN;

          
END_FUNCTION

FUNCTION assertArrayEqual_WSTRING : BOOL
  VAR_INPUT
    act : POINTER TO ARRAY[0..32000] OF WSTRING;  (* Variable to test *)
    xp : POINTER TO ARRAY[0..32000] OF WSTRING;  (* Variable to test against *)
    size : UINT;  (* Size of the array (ADR(act)) *)
  END_VAR
  VAR
    i : UINT;  (* Iterator variable *)
    vStop : UINT;  (* Size of the array / End of iteration *)
    pt1 : POINTER TO WSTRING;  (* Pointer to the element of the array act *)
    pt2 : POINTER TO WSTRING;  (* Pointer to the element of the array xp *)
  END_VAR

            vStop := (size / SIZEOF(act^[0])) - 1;

FOR i:=0 TO vStop DO
	pt1 := ADR(act^[i]);
	pt2 := ADR(xp^[i]);
	IF pt1^ <> pt2^ THEN
		assertArrayEqual_WSTRING := FALSE;
		RETURN;
	END_IF
END_FOR
(*If we reach here, all elements are equal*)
assertArrayEqual_WSTRING := TRUE;
RETURN;

          
END_FUNCTION

FUNCTION assertArrayEqual_TIME : BOOL
  VAR_INPUT
    act : POINTER TO ARRAY[0..32000] OF TIME;  (* Variable to test *)
    xp : POINTER TO ARRAY[0..32000] OF TIME;  (* Variable to test against *)
    size : UINT;  (* Size of the array (ADR(act)) *)
  END_VAR
  VAR
    i : UINT;  (* Iterator variable *)
    vStop : UINT;  (* Size of the array / End of iteration *)
    pt1 : POINTER TO TIME;  (* Pointer to the element of the array act *)
    pt2 : POINTER TO TIME;  (* Pointer to the element of the array xp *)
  END_VAR

            vStop := (size / SIZEOF(act^[0])) - 1;

FOR i:=0 TO vStop DO
	pt1 := ADR(act^[i]);
	pt2 := ADR(xp^[i]);
	IF pt1^ <> pt2^ THEN
		assertArrayEqual_TIME := FALSE;
		RETURN;
	END_IF
END_FOR
(*If we reach here, all elements are equal*)
assertArrayEqual_TIME := TRUE;
RETURN;

          
END_FUNCTION

FUNCTION assertArrayEqual_LTIME : BOOL
  VAR_INPUT
    act : POINTER TO ARRAY[0..32000] OF LTIME;  (* Variable to test *)
    xp : POINTER TO ARRAY[0..32000] OF LTIME;  (* Variable to test against *)
    size : UINT;  (* Size of the array (ADR(act)) *)
  END_VAR
  VAR
    i : UINT;  (* Iterator variable *)
    vStop : UINT;  (* Size of the array / End of iteration *)
    pt1 : POINTER TO LTIME;  (* Pointer to the element of the array act *)
    pt2 : POINTER TO LTIME;  (* Pointer to the element of the array xp *)
  END_VAR

            vStop := (size / SIZEOF(act^[0])) - 1;

FOR i:=0 TO vStop DO
	pt1 := ADR(act^[i]);
	pt2 := ADR(xp^[i]);
	IF pt1^ <> pt2^ THEN
		assertArrayEqual_LTIME := FALSE;
		RETURN;
	END_IF
END_FOR
(*If we reach here, all elements are equal*)
assertArrayEqual_LTIME := TRUE;
RETURN;

          
END_FUNCTION

FUNCTION assertArrayEqual_DATE : BOOL
  VAR_INPUT
    act : POINTER TO ARRAY[0..32000] OF DATE;  (* Variable to test *)
    xp : POINTER TO ARRAY[0..32000] OF DATE;  (* Variable to test against *)
    size : UINT;  (* Size of the array (ADR(act)) *)
  END_VAR
  VAR
    i : UINT;  (* Iterator variable *)
    vStop : UINT;  (* Size of the array / End of iteration *)
    pt1 : POINTER TO DATE;  (* Pointer to the element of the array act *)
    pt2 : POINTER TO DATE;  (* Pointer to the element of the array xp *)
  END_VAR

            vStop := (size / SIZEOF(act^[0])) - 1;

FOR i:=0 TO vStop DO
	pt1 := ADR(act^[i]);
	pt2 := ADR(xp^[i]);
	IF pt1^ <> pt2^ THEN
		assertArrayEqual_DATE := FALSE;
		RETURN;
	END_IF
END_FOR
(*If we reach here, all elements are equal*)
assertArrayEqual_DATE := TRUE;
RETURN;

          
END_FUNCTION

FUNCTION assertArrayEqual_LDATE : BOOL
  VAR_INPUT
    act : POINTER TO ARRAY[0..32000] OF LDATE;  (* Variable to test *)
    xp : POINTER TO ARRAY[0..32000] OF LDATE;  (* Variable to test against *)
    size : UINT;  (* Size of the array (ADR(act)) *)
  END_VAR
  VAR
    i : UINT;  (* Iterator variable *)
    vStop : UINT;  (* Size of the array / End of iteration *)
    pt1 : POINTER TO LDATE;  (* Pointer to the element of the array act *)
    pt2 : POINTER TO LDATE;  (* Pointer to the element of the array xp *)
  END_VAR

            vStop := (size / SIZEOF(act^[0])) - 1;

FOR i:=0 TO vStop DO
	pt1 := ADR(act^[i]);
	pt2 := ADR(xp^[i]);
	IF pt1^ <> pt2^ THEN
		assertArrayEqual_LDATE := FALSE;
		RETURN;
	END_IF
END_FOR
(*If we reach here, all elements are equal*)
assertArrayEqual_LDATE := TRUE;
RETURN;

          
END_FUNCTION

FUNCTION assertArrayEqual_DATE_AND_TIME : BOOL
  VAR_INPUT
    act : POINTER TO ARRAY[0..32000] OF DT;  (* Variable to test *)
    xp : POINTER TO ARRAY[0..32000] OF DT;  (* Variable to test against *)
    size : UINT;  (* Size of the array (ADR(act)) *)
  END_VAR
  VAR
    i : UINT;  (* Iterator variable *)
    vStop : UINT;  (* Size of the array / End of iteration *)
    pt1 : POINTER TO DT;  (* Pointer to the element of the array act *)
    pt2 : POINTER TO DT;  (* Pointer to the element of the array xp *)
  END_VAR

            vStop := (size / SIZEOF(act^[0])) - 1;

FOR i:=0 TO vStop DO
	pt1 := ADR(act^[i]);
	pt2 := ADR(xp^[i]);
	IF pt1^ <> pt2^ THEN
		assertArrayEqual_DATE_AND_TIME := FALSE;
		RETURN;
	END_IF
END_FOR
(*If we reach here, all elements are equal*)
assertArrayEqual_DATE_AND_TIME := TRUE;
RETURN;

          
END_FUNCTION

FUNCTION assertArrayEqual_LDATE_AND_TIME : BOOL
  VAR_INPUT
    act : POINTER TO ARRAY[0..32000] OF LDATE_AND_TIME;  (* Variable to test *)
    xp : POINTER TO ARRAY[0..32000] OF LDATE_AND_TIME;  (* Variable to test against *)
    size : UINT;  (* Size of the array (ADR(act)) *)
  END_VAR
  VAR
    i : UINT;  (* Iterator variable *)
    vStop : UINT;  (* Size of the array / End of iteration *)
    pt1 : POINTER TO LDATE_AND_TIME;  (* Pointer to the element of the array act *)
    pt2 : POINTER TO LDATE_AND_TIME;  (* Pointer to the element of the array xp *)
  END_VAR

            vStop := (size / SIZEOF(act^[0])) - 1;

FOR i:=0 TO vStop DO
	pt1 := ADR(act^[i]);
	pt2 := ADR(xp^[i]);
	IF pt1^ <> pt2^ THEN
		assertArrayEqual_LDATE_AND_TIME := FALSE;
		RETURN;
	END_IF
END_FOR
(*If we reach here, all elements are equal*)
assertArrayEqual_LDATE_AND_TIME := TRUE;
RETURN;

          
END_FUNCTION

FUNCTION assertArrayEqual_TIME_OF_DAY : BOOL
  VAR_INPUT
    act : POINTER TO ARRAY[0..32000] OF TOD;  (* Variable to test *)
    xp : POINTER TO ARRAY[0..32000] OF TOD;  (* Variable to test against *)
    size : UINT;  (* Size of the array (ADR(act)) *)
  END_VAR
  VAR
    i : UINT;  (* Iterator variable *)
    vStop : UINT;  (* Size of the array / End of iteration *)
    pt1 : POINTER TO TOD;  (* Pointer to the element of the array act *)
    pt2 : POINTER TO TOD;  (* Pointer to the element of the array xp *)
  END_VAR

            vStop := (size / SIZEOF(act^[0])) - 1;

FOR i:=0 TO vStop DO
	pt1 := ADR(act^[i]);
	pt2 := ADR(xp^[i]);
	IF pt1^ <> pt2^ THEN
		assertArrayEqual_TIME_OF_DAY := FALSE;
		RETURN;
	END_IF
END_FOR
(*If we reach here, all elements are equal*)
assertArrayEqual_TIME_OF_DAY := TRUE;
RETURN;

          
END_FUNCTION

FUNCTION assertArrayEqual_LTIME_OF_DAY : BOOL
  VAR_INPUT
    act : POINTER TO ARRAY[0..32000] OF LTIME_OF_DAY;  (* Variable to test *)
    xp : POINTER TO ARRAY[0..32000] OF LTIME_OF_DAY;  (* Variable to test against *)
    size : UINT;  (* Size of the array (ADR(act)) *)
  END_VAR
  VAR
    i : UINT;  (* Iterator variable *)
    vStop : UINT;  (* Size of the array / End of iteration *)
    pt1 : POINTER TO LTIME_OF_DAY;  (* Pointer to the element of the array act *)
    pt2 : POINTER TO LTIME_OF_DAY;  (* Pointer to the element of the array xp *)
  END_VAR

            vStop := (size / SIZEOF(act^[0])) - 1;

FOR i:=0 TO vStop DO
	pt1 := ADR(act^[i]);
	pt2 := ADR(xp^[i]);
	IF pt1^ <> pt2^ THEN
		assertArrayEqual_LTIME_OF_DAY := FALSE;
		RETURN;
	END_IF
END_FOR
(*If we reach here, all elements are equal*)
assertArrayEqual_LTIME_OF_DAY := TRUE;
RETURN;

          
END_FUNCTION

FUNCTION assertTrue : BOOL
  VAR_INPUT
    condition : BOOL;  (* Variable to test *)
  END_VAR

            assertTrue := condition;
RETURN;

          
END_FUNCTION

FUNCTION_BLOCK utTestSuite
  VAR_INPUT
    Id : UINT;  (* Id of the test object. Must be unique number *)
    Name : STRING(250);  (* Name of the test object *)
    RunTests : BOOL;  (* Starts all tests that are in setup state. Sets state to running. *)
    ResetTests : BOOL;  (* Sets state to setup on test cases that are PASSED or FAILED. *)
  END_VAR
  VAR_IN_OUT
    TestCases : ARRAY[0..20] OF utTestCase;  (* Array of test case definition *)
  END_VAR
  VAR_OUTPUT
    Summary : utTestCaseSummary;  (* Summary of the test results *)
  END_VAR
  VAR
    i : UINT;  (* Iterator variable *)
    runCmd : R_TRIG;  (* Trigger to prevent constant run commands *)
    resetCmd : R_TRIG;  (* Trigger to prevent constant reset commands *)
  END_VAR

            (*Copy name of object under test*)
Summary.Id := Id;
Summary.Name := Name;

(*Handle commands to start*)
runCmd(CLK:=RunTests);
resetCmd(CLK:=ResetTests);

(*Calculate total number of tests and other flags*)
Summary.TotalTests := 0;
Summary.TestsPassed := 0;
Summary.TestsFailed := 0; 
Summary.TestsRunning := FALSE;
FOR i:=0 TO 20 DO
	IF TestCases[i].id > 0 THEN
		Summary.TotalTests := Summary.TotalTests + 1;
	END_IF
	(*Start the test if the Run command is true, the test exists and it is in setup state*)
	IF TestCases[i].id > 0 AND TestCases[i].state = utTestCaseStates.SETUP AND runCmd.Q THEN
		TestCases[i].state := utTestCaseStates.RUNNING;
	END_IF
	
	(*Reset the test if the test exists and its PASSED or FAILED*)
	IF TestCases[i].id > 0 AND TestCases[i].state > utTestCaseStates.RUNNING AND resetCmd.Q THEN
		TestCases[i].state := utTestCaseStates.SETUP;
	END_IF
	
	(*Check the states of the test cases*)
	IF TestCases[i].state = utTestCaseStates.RUNNING THEN
		Summary.TestsRunning := TRUE;
	END_IF
	IF TestCases[i].state = utTestCaseStates.PASSED THEN
		Summary.TestsPassed := Summary.TestsPassed + 1;
	END_IF
	IF TestCases[i].state = utTestCaseStates.FAILED THEN
		Summary.TestsFailed := Summary.TestsFailed + 1;
	END_IF
END_FOR

(*Error if number of tests defined is 0*)
IF Summary.TotalTests = 0 THEN
	Summary.Error := utErrors.NO_TEST_CASES_DEFINED;
	RETURN;
END_IF

(*Calculate the pass rate if all tests have finished*)
IF NOT Summary.TestsRunning THEN
	Summary.PassRate := (Summary.TestsPassed / UINT_TO_REAL(Summary.TotalTests)) * 100.0;
ELSE
	Summary.PassRate := 0;
END_IF
          
END_FUNCTION_BLOCK

FUNCTION_BLOCK utTestReporter
  VAR_IN_OUT
    Results : ARRAY[0..500] OF utTestCaseSummary;  (* Summaries of tests for each POU under test *)
  END_VAR
  VAR_OUTPUT
    NrPousUnderTest : UINT;  (* Total number of POUs under test *)
    NrOfTests : UINT;  (* Total number of tests *)
    NrTestsPassed : UINT;  (* Number of tests passed *)
    NrTestsFailed : UINT;  (* Number of tests failed *)
    PassRate : REAL;  (* Total pass rate *)
    TestsInProgress : BOOL;  (* Indicates that one or more tests are in progress *)
    Error : BOOL;  (* Indicates that one or more tests are in error state *)
  END_VAR
  VAR
    i : UINT;  (* Iterator variable *)
  END_VAR

            (*Reset totals*)
NrPousUnderTest := 0;
NrOfTests := 0;
NrTestsPassed := 0;
NrTestsFailed := 0;
PassRate := 0;
TestsInProgress := FALSE;
Error := FALSE;

(*Count totals*)
FOR i:=0 TO 500 DO
	IF Results[i].Id > 0 THEN
		(*Count existing POUs under test*)
		NrPousUnderTest := NrPousUnderTest + 1;
		(*Count the pass rate. Needs to be divided in the end by the number of total tests*)
		PassRate := PassRate + Results[i].PassRate;
		(*Count the number of tests*)
		NrOfTests := NrOfTests + Results[i].TotalTests;
		(*Count the number of tests passed*)
		NrTestsPassed := NrTestsPassed + Results[i].TestsPassed;
		(*Count the number of tests failed*)
		NrTestsFailed := NrTestsFailed + Results[i].TestsFailed;
		
		(*Indicators*)
		IF Results[i].TestsRunning THEN
			TestsInProgress := TRUE;
		END_IF
		IF Results[i].Error <> utErrors.NO_ERROR THEN
			Error := TRUE;
		END_IF
	END_IF
END_FOR
PassRate := PassRate / NrPousUnderTest;
          
END_FUNCTION_BLOCK

PROGRAM test_assertNotEqual_BOOL
  VAR
    vTestCases : ARRAY[0..20] OF utTestCase;  (* Definition of all test cases for this POU *)
    testRunner : utTestSuite;  (* Test Suite fb instance to run the tests *)
    vRunAll : BOOL;  (* Manual command to run all tests for this POU *)
    vResetAll : BOOL;  (* Manual command to reset all tests for this POU *)
    vTestCase1_act : BOOL;  (* Test data 1 of test case 1 *)
    vTestCase1_xp : BOOL;  (* Test data 2 of test case 1 *)
    vTestCase2_act : BOOL;  (* Test data 1 of test case 2 *)
    vTestCase2_xp : BOOL;  (* Test data 2 of test case 2 *)
  END_VAR

                    (*Run the test cases*)
TEST_CASE_1_SETUP();
TEST_CASE_1_EXEC();

TEST_CASE_2_SETUP();
TEST_CASE_2_EXEC();

(*Instantiate the test runner*)
testRunner(
	Id := 25,
	Name := 'assertNotEqual_BOOL',
    RunTests := GVL.RunAll OR vRunAll,
	ResetTests := GVL.ResetAll OR vResetAll,
	TestCases:=vTestCases);

(*Report the results to the collection global*)
GVL.Results[testRunner.Id] := testRunner.Summary;
                  

ACTION TEST_CASE_1_SETUP:
                        IF vTestCases[0].state = utTestCaseStates.SETUP THEN
	(*Setup the test case information*)
	vTestCases[0].id := 1;
	vTestCases[0].desc[0] := 'RETURNS TRUE WHEN PARAMETERS NOT EQUAL';
    vTestCases[0].desc[1] := 'Tests if the function returns True if the passed in parameters do not hold the same value';
	vTestCases[0].desc[2] := 'PASS IF: Return value is TRUE';
	
	(*Setup needed variables*)
	vTestCase1_act := TRUE;
	vTestCase1_xp := FALSE;
END_IF
                      
END_ACTION

ACTION TEST_CASE_1_EXEC:
                        IF vTestCases[0].state = utTestCaseStates.RUNNING THEN
	(*Run the test case*)
	IF assertNotEqual_BOOL(vTestCase1_act, vTestCase1_xp) THEN
		vTestCases[0].state := utTestCaseStates.PASSED;
		vTestCases[0].msg := 'Passed parameters were not equal and function returned TRUE -> PASS';
	ELSE
		vTestCases[0].state := utTestCaseStates.FAILED;
		vTestCases[0].msg := 'Passed parameters were not equal and function returned FALSE -> FAIL';
	END_IF
END_IF
                      
END_ACTION

ACTION TEST_CASE_2_SETUP:
                        IF vTestCases[1].state = utTestCaseStates.SETUP THEN
	(*Setup the test case information*)
	vTestCases[1].id := 2;
	vTestCases[1].desc[0] := 'RETURNS FALSE WHEN PARAMETERS EQUAL';
    vTestCases[1].desc[1] := 'Tests if the function returns False if the passed in parameters hold the same value';
	vTestCases[1].desc[2] := 'PASS IF: Return value is FALSE';
	
	(*Setup needed variables*)
	vTestCase2_act := TRUE;
	vTestCase2_xp := TRUE;
END_IF
                      
END_ACTION

ACTION TEST_CASE_2_EXEC:
                        IF vTestCases[1].state = utTestCaseStates.RUNNING THEN
	(*Run the test case*)
	IF NOT assertNotEqual_BOOL(vTestCase2_act, vTestCase2_xp) THEN
		vTestCases[1].state := utTestCaseStates.PASSED;
		vTestCases[1].msg := 'Passed parameters were equal and function returned FALSE -> PASS';
	ELSE
		vTestCases[1].state := utTestCaseStates.FAILED;
		vTestCases[1].msg := 'Passed parameters were equal and function returned TRUE -> FAIL';
	END_IF
END_IF
                      
END_ACTION
END_PROGRAM

PROGRAM test_assertNotEqual_INT
  VAR
    vTestCases : ARRAY[0..20] OF utTestCase;  (* Definition of all test cases for this POU *)
    testRunner : utTestSuite;  (* Test Suite fb instance to run the tests *)
    vRunAll : BOOL;  (* Manual command to run all tests for this POU *)
    vResetAll : BOOL;  (* Manual command to reset all tests for this POU *)
    vTestCase1_act : INT;  (* Test data 1 of test case 1 *)
    vTestCase1_xp : INT;  (* Test data 2 of test case 1 *)
    vTestCase2_act : INT;  (* Test data 1 of test case 2 *)
    vTestCase2_xp : INT;  (* Test data 2 of test case 2 *)
  END_VAR

                    (*Run the test cases*)
TEST_CASE_1_SETUP();
TEST_CASE_1_EXEC();

TEST_CASE_2_SETUP();
TEST_CASE_2_EXEC();

(*Instantiate the test runner*)
testRunner(
	Id := 32,
	Name := 'assertNotEqual_INT',
    RunTests := GVL.RunAll OR vRunAll,
	ResetTests := GVL.ResetAll OR vResetAll,
	TestCases:=vTestCases);

(*Report the results to the collection global*)
GVL.Results[testRunner.Id] := testRunner.Summary;
                  

ACTION TEST_CASE_1_SETUP:
                        IF vTestCases[0].state = utTestCaseStates.SETUP THEN
	(*Setup the test case information*)
	vTestCases[0].id := 1;
	vTestCases[0].desc[0] := 'RETURNS TRUE WHEN PARAMETERS NOT EQUAL';
    vTestCases[0].desc[1] := 'Tests if the function returns True if the passed in parameters do not hold the same value';
	vTestCases[0].desc[2] := 'PASS IF: Return value is TRUE';
	
	(*Setup needed variables*)
	vTestCase1_act := REAL_TO_INT(115.4);
	vTestCase1_xp := REAL_TO_INT(-85.4);
END_IF
                      
END_ACTION

ACTION TEST_CASE_1_EXEC:
                        IF vTestCases[0].state = utTestCaseStates.RUNNING THEN
	(*Run the test case*)
	IF assertNotEqual_INT(vTestCase1_act, vTestCase1_xp) THEN
		vTestCases[0].state := utTestCaseStates.PASSED;
		vTestCases[0].msg := 'Passed parameters were not equal and function returned TRUE -> PASS';
	ELSE
		vTestCases[0].state := utTestCaseStates.FAILED;
		vTestCases[0].msg := 'Passed parameters were not equal and function returned FALSE -> FAIL';
	END_IF
END_IF
                      
END_ACTION

ACTION TEST_CASE_2_SETUP:
                        IF vTestCases[1].state = utTestCaseStates.SETUP THEN
	(*Setup the test case information*)
	vTestCases[1].id := 2;
	vTestCases[1].desc[0] := 'RETURNS FALSE WHEN PARAMETERS EQUAL';
    vTestCases[1].desc[1] := 'Tests if the function returns False if the passed in parameters hold the same value';
	vTestCases[1].desc[2] := 'PASS IF: Return value is FALSE';
	
	(*Setup needed variables*)
	vTestCase2_act := REAL_TO_INT(115.4);
	vTestCase2_xp := REAL_TO_INT(115.4);
END_IF
                      
END_ACTION

ACTION TEST_CASE_2_EXEC:
                        IF vTestCases[1].state = utTestCaseStates.RUNNING THEN
	(*Run the test case*)
	IF NOT assertNotEqual_INT(vTestCase2_act, vTestCase2_xp) THEN
		vTestCases[1].state := utTestCaseStates.PASSED;
		vTestCases[1].msg := 'Passed parameters were equal and function returned FALSE -> PASS';
	ELSE
		vTestCases[1].state := utTestCaseStates.FAILED;
		vTestCases[1].msg := 'Passed parameters were equal and function returned TRUE -> FAIL';
	END_IF
END_IF
                      
END_ACTION
END_PROGRAM

PROGRAM test_assertNotEqual_DATE_AND_TIME
  VAR
    vTestCases : ARRAY[0..20] OF utTestCase;  (* Definition of all test cases for this POU *)
    testRunner : utTestSuite;  (* Test Suite fb instance to run the tests *)
    vRunAll : BOOL;  (* Manual command to run all tests for this POU *)
    vResetAll : BOOL;  (* Manual command to reset all tests for this POU *)
    vTestCase1_act : DT;  (* Test data 1 of test case 1 *)
    vTestCase1_xp : DT;  (* Test data 2 of test case 1 *)
    vTestCase2_act : DT;  (* Test data 1 of test case 2 *)
    vTestCase2_xp : DT;  (* Test data 2 of test case 2 *)
  END_VAR

                    (*Run the test cases*)
TEST_CASE_1_SETUP();
TEST_CASE_1_EXEC();

TEST_CASE_2_SETUP();
TEST_CASE_2_EXEC();

(*Instantiate the test runner*)
testRunner(
	Id := 46,
	Name := 'assertNotEqual_DATE_AND_TIME',
    RunTests := GVL.RunAll OR vRunAll,
	ResetTests := GVL.ResetAll OR vResetAll,
	TestCases:=vTestCases);

(*Report the results to the collection global*)
GVL.Results[testRunner.Id] := testRunner.Summary;
                  

ACTION TEST_CASE_1_SETUP:
                        IF vTestCases[0].state = utTestCaseStates.SETUP THEN
	(*Setup the test case information*)
	vTestCases[0].id := 1;
	vTestCases[0].desc[0] := 'RETURNS TRUE WHEN PARAMETERS NOT EQUAL';
    vTestCases[0].desc[1] := 'Tests if the function returns True if the passed in parameters do not hold the same value';
	vTestCases[0].desc[2] := 'PASS IF: Return value is TRUE';
	
	(*Setup needed variables*)
	vTestCase1_act := REAL_TO_DT(115.4);
	vTestCase1_xp := REAL_TO_DT(-85.4);
END_IF
                      
END_ACTION

ACTION TEST_CASE_1_EXEC:
                        IF vTestCases[0].state = utTestCaseStates.RUNNING THEN
	(*Run the test case*)
	IF assertNotEqual_DATE_AND_TIME(vTestCase1_act, vTestCase1_xp) THEN
		vTestCases[0].state := utTestCaseStates.PASSED;
		vTestCases[0].msg := 'Passed parameters were not equal and function returned TRUE -> PASS';
	ELSE
		vTestCases[0].state := utTestCaseStates.FAILED;
		vTestCases[0].msg := 'Passed parameters were not equal and function returned FALSE -> FAIL';
	END_IF
END_IF
                      
END_ACTION

ACTION TEST_CASE_2_SETUP:
                        IF vTestCases[1].state = utTestCaseStates.SETUP THEN
	(*Setup the test case information*)
	vTestCases[1].id := 2;
	vTestCases[1].desc[0] := 'RETURNS FALSE WHEN PARAMETERS EQUAL';
    vTestCases[1].desc[1] := 'Tests if the function returns False if the passed in parameters hold the same value';
	vTestCases[1].desc[2] := 'PASS IF: Return value is FALSE';
	
	(*Setup needed variables*)
	vTestCase2_act := REAL_TO_DT(115.4);
	vTestCase2_xp := REAL_TO_DT(115.4);
END_IF
                      
END_ACTION

ACTION TEST_CASE_2_EXEC:
                        IF vTestCases[1].state = utTestCaseStates.RUNNING THEN
	(*Run the test case*)
	IF NOT assertNotEqual_DATE_AND_TIME(vTestCase2_act, vTestCase2_xp) THEN
		vTestCases[1].state := utTestCaseStates.PASSED;
		vTestCases[1].msg := 'Passed parameters were equal and function returned FALSE -> PASS';
	ELSE
		vTestCases[1].state := utTestCaseStates.FAILED;
		vTestCases[1].msg := 'Passed parameters were equal and function returned TRUE -> FAIL';
	END_IF
END_IF
                      
END_ACTION
END_PROGRAM

PROGRAM test_assertGreater_LWORD
  VAR
    vTestCases : ARRAY[0..20] OF utTestCase;  (* Definition of all test cases for this POU *)
    testRunner : utTestSuite;  (* Test Suite fb instance to run the tests *)
    vRunAll : BOOL;  (* Manual command to run all tests for this POU *)
    vResetAll : BOOL;  (* Manual command to reset all tests for this POU *)
    vTestCase1_act : LWORD;  (* Test data 1 of test case 1 *)
    vTestCase1_xp : LWORD;  (* Test data 2 of test case 1 *)
    vTestCase2_act : LWORD;  (* Test data 1 of test case 2 *)
    vTestCase2_xp : LWORD;  (* Test data 2 of test case 2 *)
  END_VAR

                    (*Run the test cases*)
TEST_CASE_1_SETUP();
TEST_CASE_1_EXEC();

TEST_CASE_2_SETUP();
TEST_CASE_2_EXEC();

(*Instantiate the test runner*)
testRunner(
	Id := 53,
	Name := 'assertGreater_LWORD',
    RunTests := GVL.RunAll OR vRunAll,
	ResetTests := GVL.ResetAll OR vResetAll,
	TestCases:=vTestCases);

(*Report the results to the collection global*)
GVL.Results[testRunner.Id] := testRunner.Summary;
                  

ACTION TEST_CASE_1_SETUP:
                        IF vTestCases[0].state = utTestCaseStates.SETUP THEN
	(*Setup the test case information*)
	vTestCases[0].id := 1;
	vTestCases[0].desc[0] := 'RETURNS TRUE WHEN PARAMETER ACT GREATER THAN XP';
    vTestCases[0].desc[1] := 'Tests if the function returns True if the parameter act is greater than parameter xp';
	vTestCases[0].desc[2] := 'PASS IF: Return value is TRUE';
	
	(*Setup needed variables*)
	vTestCase1_act := REAL_TO_LWORD(115.4);
	vTestCase1_xp := REAL_TO_LWORD(85.4);
END_IF
                      
END_ACTION

ACTION TEST_CASE_1_EXEC:
                        IF vTestCases[0].state = utTestCaseStates.RUNNING THEN
	(*Run the test case*)
	IF assertGreater_LWORD(vTestCase1_act, vTestCase1_xp) THEN
		vTestCases[0].state := utTestCaseStates.PASSED;
		vTestCases[0].msg := 'Parameter act was greater than xp and function returned TRUE -> PASS';
	ELSE
		vTestCases[0].state := utTestCaseStates.FAILED;
		vTestCases[0].msg := 'Parameter act was greater than xp and function returned FALSE -> FAIL';
	END_IF
END_IF
                      
END_ACTION

ACTION TEST_CASE_2_SETUP:
                        IF vTestCases[1].state = utTestCaseStates.SETUP THEN
	(*Setup the test case information*)
	vTestCases[1].id := 2;
    vTestCases[1].desc[0] := 'RETURNS FALSE WHEN PARAMETER ACT LESS THAN XP';
    vTestCases[1].desc[1] := 'Tests if the function returns False if the parameter act is less than parameter xp';
	vTestCases[1].desc[2] := 'PASS IF: Return value is FALSE';
	
	(*Setup needed variables*)
	vTestCase2_act := REAL_TO_LWORD(8.4);
	vTestCase2_xp := REAL_TO_LWORD(85.4);
END_IF
                      
END_ACTION

ACTION TEST_CASE_2_EXEC:
                        IF vTestCases[1].state = utTestCaseStates.RUNNING THEN
	(*Run the test case*)
	IF NOT assertGreater_LWORD(vTestCase2_act, vTestCase2_xp) THEN
		vTestCases[1].state := utTestCaseStates.PASSED;
		vTestCases[1].msg := 'Parameter act was less than xp and function returned FALSE -> PASS';
	ELSE
		vTestCases[1].state := utTestCaseStates.FAILED;
		vTestCases[1].msg := 'Parameter act was less than xp and function returned TRUE -> FAIL';
	END_IF
END_IF
                      
END_ACTION
END_PROGRAM

PROGRAM test_assertNotEqual_LREAL
  VAR
    vTestCases : ARRAY[0..20] OF utTestCase;  (* Definition of all test cases for this POU *)
    testRunner : utTestSuite;  (* Test Suite fb instance to run the tests *)
    vRunAll : BOOL;  (* Manual command to run all tests for this POU *)
    vResetAll : BOOL;  (* Manual command to reset all tests for this POU *)
    vTestCase1_act : LREAL;  (* Test data 1 of test case 1 *)
    vTestCase1_xp : LREAL;  (* Test data 2 of test case 1 *)
    vTestCase2_act : LREAL;  (* Test data 1 of test case 2 *)
    vTestCase2_xp : LREAL;  (* Test data 2 of test case 2 *)
  END_VAR

                    (*Run the test cases*)
TEST_CASE_1_SETUP();
TEST_CASE_1_EXEC();

TEST_CASE_2_SETUP();
TEST_CASE_2_EXEC();

(*Instantiate the test runner*)
testRunner(
	Id := 39,
	Name := 'assertNotEqual_LREAL',
    RunTests := GVL.RunAll OR vRunAll,
	ResetTests := GVL.ResetAll OR vResetAll,
	TestCases:=vTestCases);

(*Report the results to the collection global*)
GVL.Results[testRunner.Id] := testRunner.Summary;
                  

ACTION TEST_CASE_1_SETUP:
                        IF vTestCases[0].state = utTestCaseStates.SETUP THEN
	(*Setup the test case information*)
	vTestCases[0].id := 1;
	vTestCases[0].desc[0] := 'RETURNS TRUE WHEN PARAMETERS NOT EQUAL';
    vTestCases[0].desc[1] := 'Tests if the function returns True if the passed in parameters do not hold the same value';
	vTestCases[0].desc[2] := 'PASS IF: Return value is TRUE';
	
	(*Setup needed variables*)
	vTestCase1_act := REAL_TO_LREAL(115.4);
	vTestCase1_xp := REAL_TO_LREAL(-85.4);
END_IF
                      
END_ACTION

ACTION TEST_CASE_1_EXEC:
                        IF vTestCases[0].state = utTestCaseStates.RUNNING THEN
	(*Run the test case*)
	IF assertNotEqual_LREAL(vTestCase1_act, vTestCase1_xp) THEN
		vTestCases[0].state := utTestCaseStates.PASSED;
		vTestCases[0].msg := 'Passed parameters were not equal and function returned TRUE -> PASS';
	ELSE
		vTestCases[0].state := utTestCaseStates.FAILED;
		vTestCases[0].msg := 'Passed parameters were not equal and function returned FALSE -> FAIL';
	END_IF
END_IF
                      
END_ACTION

ACTION TEST_CASE_2_SETUP:
                        IF vTestCases[1].state = utTestCaseStates.SETUP THEN
	(*Setup the test case information*)
	vTestCases[1].id := 2;
	vTestCases[1].desc[0] := 'RETURNS FALSE WHEN PARAMETERS EQUAL';
    vTestCases[1].desc[1] := 'Tests if the function returns False if the passed in parameters hold the same value';
	vTestCases[1].desc[2] := 'PASS IF: Return value is FALSE';
	
	(*Setup needed variables*)
	vTestCase2_act := REAL_TO_LREAL(115.4);
	vTestCase2_xp := REAL_TO_LREAL(115.4);
END_IF
                      
END_ACTION

ACTION TEST_CASE_2_EXEC:
                        IF vTestCases[1].state = utTestCaseStates.RUNNING THEN
	(*Run the test case*)
	IF NOT assertNotEqual_LREAL(vTestCase2_act, vTestCase2_xp) THEN
		vTestCases[1].state := utTestCaseStates.PASSED;
		vTestCases[1].msg := 'Passed parameters were equal and function returned FALSE -> PASS';
	ELSE
		vTestCases[1].state := utTestCaseStates.FAILED;
		vTestCases[1].msg := 'Passed parameters were equal and function returned TRUE -> FAIL';
	END_IF
END_IF
                      
END_ACTION
END_PROGRAM

PROGRAM test_assertLess_LTIME
  VAR
    vTestCases : ARRAY[0..20] OF utTestCase;  (* Definition of all test cases for this POU *)
    testRunner : utTestSuite;  (* Test Suite fb instance to run the tests *)
    vRunAll : BOOL;  (* Manual command to run all tests for this POU *)
    vResetAll : BOOL;  (* Manual command to reset all tests for this POU *)
    vTestCase1_act : LTIME;  (* Test data 1 of test case 1 *)
    vTestCase1_xp : LTIME;  (* Test data 2 of test case 1 *)
    vTestCase2_act : LTIME;  (* Test data 1 of test case 2 *)
    vTestCase2_xp : LTIME;  (* Test data 2 of test case 2 *)
  END_VAR

                    (*Run the test cases*)
TEST_CASE_1_SETUP();
TEST_CASE_1_EXEC();

TEST_CASE_2_SETUP();
TEST_CASE_2_EXEC();

(*Instantiate the test runner*)
testRunner(
	Id := 109,
	Name := 'assertLess_LTIME',
    RunTests := GVL.RunAll OR vRunAll,
	ResetTests := GVL.ResetAll OR vResetAll,
	TestCases:=vTestCases);

(*Report the results to the collection global*)
GVL.Results[testRunner.Id] := testRunner.Summary;
                  

ACTION TEST_CASE_1_SETUP:
                        IF vTestCases[0].state = utTestCaseStates.SETUP THEN
	(*Setup the test case information*)
	vTestCases[0].id := 1;
	vTestCases[0].desc[0] := 'RETURNS TRUE WHEN PARAMETER ACT LESS THAN XP';
    vTestCases[0].desc[1] := 'Tests if the function returns True if the parameter act is less than parameter xp';
	vTestCases[0].desc[2] := 'PASS IF: Return value is TRUE';
	
	(*Setup needed variables*)
	vTestCase1_act := REAL_TO_LTIME(85.4);
	vTestCase1_xp := REAL_TO_LTIME(115.4);
END_IF
                      
END_ACTION

ACTION TEST_CASE_1_EXEC:
                        IF vTestCases[0].state = utTestCaseStates.RUNNING THEN
	(*Run the test case*)
	IF assertLess_LTIME(vTestCase1_act, vTestCase1_xp) THEN
		vTestCases[0].state := utTestCaseStates.PASSED;
		vTestCases[0].msg := 'Parameter act was less than xp and function returned TRUE -> PASS';
	ELSE
		vTestCases[0].state := utTestCaseStates.FAILED;
		vTestCases[0].msg := 'Parameter act was less than xp and function returned FALSE -> FAIL';
	END_IF
END_IF
                      
END_ACTION

ACTION TEST_CASE_2_SETUP:
                        IF vTestCases[1].state = utTestCaseStates.SETUP THEN
	(*Setup the test case information*)
	vTestCases[1].id := 2;
    vTestCases[1].desc[0] := 'RETURNS FALSE WHEN PARAMETER ACT GREATER THAN XP';
    vTestCases[1].desc[1] := 'Tests if the function returns False if the parameter act is greater than parameter xp';
	vTestCases[1].desc[2] := 'PASS IF: Return value is FALSE';
	
	(*Setup needed variables*)
	vTestCase2_act := REAL_TO_LTIME(115.4);
	vTestCase2_xp := REAL_TO_LTIME(85.4);
END_IF
                      
END_ACTION

ACTION TEST_CASE_2_EXEC:
                        IF vTestCases[1].state = utTestCaseStates.RUNNING THEN
	(*Run the test case*)
	IF NOT assertLess_LTIME(vTestCase2_act, vTestCase2_xp) THEN
		vTestCases[1].state := utTestCaseStates.PASSED;
		vTestCases[1].msg := 'Parameter act was greater than xp and function returned FALSE -> PASS';
	ELSE
		vTestCases[1].state := utTestCaseStates.FAILED;
		vTestCases[1].msg := 'Parameter act was greater than xp and function returned TRUE -> FAIL';
	END_IF
END_IF
                      
END_ACTION
END_PROGRAM

PROGRAM test_assertLessEqual_BYTE
  VAR
    vTestCases : ARRAY[0..20] OF utTestCase;  (* Definition of all test cases for this POU *)
    testRunner : utTestSuite;  (* Test Suite fb instance to run the tests *)
    vRunAll : BOOL;  (* Manual command to run all tests for this POU *)
    vResetAll : BOOL;  (* Manual command to reset all tests for this POU *)
    vTestCase1_act : BYTE;  (* Test data 1 of test case 1 *)
    vTestCase1_xp : BYTE;  (* Test data 2 of test case 1 *)
    vTestCase2_act : BYTE;  (* Test data 1 of test case 2 *)
    vTestCase2_xp : BYTE;  (* Test data 2 of test case 2 *)
    vTestCase3_act : BYTE;  (* Test data 1 of test case 3 *)
    vTestCase3_xp : BYTE;  (* Test data 2 of test case 3 *)
  END_VAR

                    (*Run the test cases*)
TEST_CASE_1_SETUP();
TEST_CASE_1_EXEC();

TEST_CASE_2_SETUP();
TEST_CASE_2_EXEC();

TEST_CASE_3_SETUP();
TEST_CASE_3_EXEC();

(*Instantiate the test runner*)
testRunner(
	Id := 116,
	Name := 'assertLessEqual_BYTE',
    RunTests := GVL.RunAll OR vRunAll,
	ResetTests := GVL.ResetAll OR vResetAll,
	TestCases:=vTestCases);

(*Report the results to the collection global*)
GVL.Results[testRunner.Id] := testRunner.Summary;
                  

ACTION TEST_CASE_1_SETUP:
                        IF vTestCases[0].state = utTestCaseStates.SETUP THEN
	(*Setup the test case information*)
	vTestCases[0].id := 1;
	vTestCases[0].desc[0] := 'RETURNS TRUE WHEN PARAMETER ACT LESS THAN XP';
    vTestCases[0].desc[1] := 'Tests if the function returns True if the parameter act is less than parameter xp';
	vTestCases[0].desc[2] := 'PASS IF: Return value is TRUE';
	
	(*Setup needed variables*)
	vTestCase1_act := REAL_TO_BYTE(85.4);
	vTestCase1_xp := REAL_TO_BYTE(115.4);
END_IF
                      
END_ACTION

ACTION TEST_CASE_1_EXEC:
                        IF vTestCases[0].state = utTestCaseStates.RUNNING THEN
	(*Run the test case*)
	IF assertLessEqual_BYTE(vTestCase1_act, vTestCase1_xp) THEN
		vTestCases[0].state := utTestCaseStates.PASSED;
		vTestCases[0].msg := 'Parameter act was less than xp and function returned TRUE -> PASS';
	ELSE
		vTestCases[0].state := utTestCaseStates.FAILED;
		vTestCases[0].msg := 'Parameter act was less than xp and function returned FALSE -> FAIL';
	END_IF
END_IF
                      
END_ACTION

ACTION TEST_CASE_2_SETUP:
                        IF vTestCases[1].state = utTestCaseStates.SETUP THEN
	(*Setup the test case information*)
	vTestCases[1].id := 2;
    vTestCases[1].desc[0] := 'RETURNS TRUE WHEN PARAMETER ACT EQUAL TO XP';
    vTestCases[1].desc[1] := 'Tests if the function returns True if the parameter act is equal to parameter xp';
	vTestCases[1].desc[2] := 'PASS IF: Return value is TRUE';
	
	(*Setup needed variables*)
	vTestCase2_act := REAL_TO_BYTE(115.4);
	vTestCase2_xp := REAL_TO_BYTE(115.4);
END_IF
                      
END_ACTION

ACTION TEST_CASE_2_EXEC:
                        IF vTestCases[1].state = utTestCaseStates.RUNNING THEN
	(*Run the test case*)
	IF assertLessEqual_BYTE(vTestCase2_act, vTestCase2_xp) THEN
		vTestCases[1].state := utTestCaseStates.PASSED;
		vTestCases[1].msg := 'Parameter act was equal to xp and function returned TRUE -> PASS';
	ELSE
		vTestCases[1].state := utTestCaseStates.FAILED;
		vTestCases[1].msg := 'Parameter act was equal to xp and function returned FALSE -> FAIL';
	END_IF
END_IF
                      
END_ACTION

ACTION TEST_CASE_3_SETUP:
                        IF vTestCases[2].state = utTestCaseStates.SETUP THEN
	(*Setup the test case information*)
	vTestCases[2].id := 3;
    vTestCases[2].desc[0] := 'RETURNS FALSE WHEN PARAMETER ACT GREATER THAN XP';
    vTestCases[2].desc[1] := 'Tests if the function returns False if the parameter act is greater than parameter xp';
	vTestCases[2].desc[2] := 'PASS IF: Return value is FALSE';
	
	(*Setup needed variables*)
	vTestCase3_act := REAL_TO_BYTE(115.4);
	vTestCase3_xp := REAL_TO_BYTE(85.4);
END_IF
                      
END_ACTION

ACTION TEST_CASE_3_EXEC:
                        IF vTestCases[2].state = utTestCaseStates.RUNNING THEN
	(*Run the test case*)
	IF NOT assertLessEqual_BYTE(vTestCase3_act, vTestCase3_xp) THEN
		vTestCases[2].state := utTestCaseStates.PASSED;
		vTestCases[2].msg := 'Parameter act was greater than xp and function returned FALSE -> PASS';
	ELSE
		vTestCases[2].state := utTestCaseStates.FAILED;
		vTestCases[2].msg := 'Parameter act was greater than xp and function returned TRUE -> FAIL';
	END_IF
END_IF
                      
END_ACTION
END_PROGRAM

PROGRAM test_assertLess_WORD
  VAR
    vTestCases : ARRAY[0..20] OF utTestCase;  (* Definition of all test cases for this POU *)
    testRunner : utTestSuite;  (* Test Suite fb instance to run the tests *)
    vRunAll : BOOL;  (* Manual command to run all tests for this POU *)
    vResetAll : BOOL;  (* Manual command to reset all tests for this POU *)
    vTestCase1_act : WORD;  (* Test data 1 of test case 1 *)
    vTestCase1_xp : WORD;  (* Test data 2 of test case 1 *)
    vTestCase2_act : WORD;  (* Test data 1 of test case 2 *)
    vTestCase2_xp : WORD;  (* Test data 2 of test case 2 *)
  END_VAR

                    (*Run the test cases*)
TEST_CASE_1_SETUP();
TEST_CASE_1_EXEC();

TEST_CASE_2_SETUP();
TEST_CASE_2_EXEC();

(*Instantiate the test runner*)
testRunner(
	Id := 95,
	Name := 'assertLess_WORD',
    RunTests := GVL.RunAll OR vRunAll,
	ResetTests := GVL.ResetAll OR vResetAll,
	TestCases:=vTestCases);

(*Report the results to the collection global*)
GVL.Results[testRunner.Id] := testRunner.Summary;
                  

ACTION TEST_CASE_1_SETUP:
                        IF vTestCases[0].state = utTestCaseStates.SETUP THEN
	(*Setup the test case information*)
	vTestCases[0].id := 1;
	vTestCases[0].desc[0] := 'RETURNS TRUE WHEN PARAMETER ACT LESS THAN XP';
    vTestCases[0].desc[1] := 'Tests if the function returns True if the parameter act is less than parameter xp';
	vTestCases[0].desc[2] := 'PASS IF: Return value is TRUE';
	
	(*Setup needed variables*)
	vTestCase1_act := REAL_TO_WORD(85.4);
	vTestCase1_xp := REAL_TO_WORD(115.4);
END_IF
                      
END_ACTION

ACTION TEST_CASE_1_EXEC:
                        IF vTestCases[0].state = utTestCaseStates.RUNNING THEN
	(*Run the test case*)
	IF assertLess_WORD(vTestCase1_act, vTestCase1_xp) THEN
		vTestCases[0].state := utTestCaseStates.PASSED;
		vTestCases[0].msg := 'Parameter act was less than xp and function returned TRUE -> PASS';
	ELSE
		vTestCases[0].state := utTestCaseStates.FAILED;
		vTestCases[0].msg := 'Parameter act was less than xp and function returned FALSE -> FAIL';
	END_IF
END_IF
                      
END_ACTION

ACTION TEST_CASE_2_SETUP:
                        IF vTestCases[1].state = utTestCaseStates.SETUP THEN
	(*Setup the test case information*)
	vTestCases[1].id := 2;
    vTestCases[1].desc[0] := 'RETURNS FALSE WHEN PARAMETER ACT GREATER THAN XP';
    vTestCases[1].desc[1] := 'Tests if the function returns False if the parameter act is greater than parameter xp';
	vTestCases[1].desc[2] := 'PASS IF: Return value is FALSE';
	
	(*Setup needed variables*)
	vTestCase2_act := REAL_TO_WORD(115.4);
	vTestCase2_xp := REAL_TO_WORD(85.4);
END_IF
                      
END_ACTION

ACTION TEST_CASE_2_EXEC:
                        IF vTestCases[1].state = utTestCaseStates.RUNNING THEN
	(*Run the test case*)
	IF NOT assertLess_WORD(vTestCase2_act, vTestCase2_xp) THEN
		vTestCases[1].state := utTestCaseStates.PASSED;
		vTestCases[1].msg := 'Parameter act was greater than xp and function returned FALSE -> PASS';
	ELSE
		vTestCases[1].state := utTestCaseStates.FAILED;
		vTestCases[1].msg := 'Parameter act was greater than xp and function returned TRUE -> FAIL';
	END_IF
END_IF
                      
END_ACTION
END_PROGRAM

PROGRAM test_assertLess_DINT
  VAR
    vTestCases : ARRAY[0..20] OF utTestCase;  (* Definition of all test cases for this POU *)
    testRunner : utTestSuite;  (* Test Suite fb instance to run the tests *)
    vRunAll : BOOL;  (* Manual command to run all tests for this POU *)
    vResetAll : BOOL;  (* Manual command to reset all tests for this POU *)
    vTestCase1_act : DINT;  (* Test data 1 of test case 1 *)
    vTestCase1_xp : DINT;  (* Test data 2 of test case 1 *)
    vTestCase2_act : DINT;  (* Test data 1 of test case 2 *)
    vTestCase2_xp : DINT;  (* Test data 2 of test case 2 *)
  END_VAR

                    (*Run the test cases*)
TEST_CASE_1_SETUP();
TEST_CASE_1_EXEC();

TEST_CASE_2_SETUP();
TEST_CASE_2_EXEC();

(*Instantiate the test runner*)
testRunner(
	Id := 102,
	Name := 'assertLess_DINT',
    RunTests := GVL.RunAll OR vRunAll,
	ResetTests := GVL.ResetAll OR vResetAll,
	TestCases:=vTestCases);

(*Report the results to the collection global*)
GVL.Results[testRunner.Id] := testRunner.Summary;
                  

ACTION TEST_CASE_1_SETUP:
                        IF vTestCases[0].state = utTestCaseStates.SETUP THEN
	(*Setup the test case information*)
	vTestCases[0].id := 1;
	vTestCases[0].desc[0] := 'RETURNS TRUE WHEN PARAMETER ACT LESS THAN XP';
    vTestCases[0].desc[1] := 'Tests if the function returns True if the parameter act is less than parameter xp';
	vTestCases[0].desc[2] := 'PASS IF: Return value is TRUE';
	
	(*Setup needed variables*)
	vTestCase1_act := REAL_TO_DINT(85.4);
	vTestCase1_xp := REAL_TO_DINT(115.4);
END_IF
                      
END_ACTION

ACTION TEST_CASE_1_EXEC:
                        IF vTestCases[0].state = utTestCaseStates.RUNNING THEN
	(*Run the test case*)
	IF assertLess_DINT(vTestCase1_act, vTestCase1_xp) THEN
		vTestCases[0].state := utTestCaseStates.PASSED;
		vTestCases[0].msg := 'Parameter act was less than xp and function returned TRUE -> PASS';
	ELSE
		vTestCases[0].state := utTestCaseStates.FAILED;
		vTestCases[0].msg := 'Parameter act was less than xp and function returned FALSE -> FAIL';
	END_IF
END_IF
                      
END_ACTION

ACTION TEST_CASE_2_SETUP:
                        IF vTestCases[1].state = utTestCaseStates.SETUP THEN
	(*Setup the test case information*)
	vTestCases[1].id := 2;
    vTestCases[1].desc[0] := 'RETURNS FALSE WHEN PARAMETER ACT GREATER THAN XP';
    vTestCases[1].desc[1] := 'Tests if the function returns False if the parameter act is greater than parameter xp';
	vTestCases[1].desc[2] := 'PASS IF: Return value is FALSE';
	
	(*Setup needed variables*)
	vTestCase2_act := REAL_TO_DINT(115.4);
	vTestCase2_xp := REAL_TO_DINT(85.4);
END_IF
                      
END_ACTION

ACTION TEST_CASE_2_EXEC:
                        IF vTestCases[1].state = utTestCaseStates.RUNNING THEN
	(*Run the test case*)
	IF NOT assertLess_DINT(vTestCase2_act, vTestCase2_xp) THEN
		vTestCases[1].state := utTestCaseStates.PASSED;
		vTestCases[1].msg := 'Parameter act was greater than xp and function returned FALSE -> PASS';
	ELSE
		vTestCases[1].state := utTestCaseStates.FAILED;
		vTestCases[1].msg := 'Parameter act was greater than xp and function returned TRUE -> FAIL';
	END_IF
END_IF
                      
END_ACTION
END_PROGRAM

PROGRAM test_assertGreater_LDATE
  VAR
    vTestCases : ARRAY[0..20] OF utTestCase;  (* Definition of all test cases for this POU *)
    testRunner : utTestSuite;  (* Test Suite fb instance to run the tests *)
    vRunAll : BOOL;  (* Manual command to run all tests for this POU *)
    vResetAll : BOOL;  (* Manual command to reset all tests for this POU *)
    vTestCase1_act : LDATE;  (* Test data 1 of test case 1 *)
    vTestCase1_xp : LDATE;  (* Test data 2 of test case 1 *)
    vTestCase2_act : LDATE;  (* Test data 1 of test case 2 *)
    vTestCase2_xp : LDATE;  (* Test data 2 of test case 2 *)
  END_VAR

                    (*Run the test cases*)
TEST_CASE_1_SETUP();
TEST_CASE_1_EXEC();

TEST_CASE_2_SETUP();
TEST_CASE_2_EXEC();

(*Instantiate the test runner*)
testRunner(
	Id := 67,
	Name := 'assertGreater_LDATE',
    RunTests := GVL.RunAll OR vRunAll,
	ResetTests := GVL.ResetAll OR vResetAll,
	TestCases:=vTestCases);

(*Report the results to the collection global*)
GVL.Results[testRunner.Id] := testRunner.Summary;
                  

ACTION TEST_CASE_1_SETUP:
                        IF vTestCases[0].state = utTestCaseStates.SETUP THEN
	(*Setup the test case information*)
	vTestCases[0].id := 1;
	vTestCases[0].desc[0] := 'RETURNS TRUE WHEN PARAMETER ACT GREATER THAN XP';
    vTestCases[0].desc[1] := 'Tests if the function returns True if the parameter act is greater than parameter xp';
	vTestCases[0].desc[2] := 'PASS IF: Return value is TRUE';
	
	(*Setup needed variables*)
	vTestCase1_act := REAL_TO_LDATE(115.4);
	vTestCase1_xp := REAL_TO_LDATE(85.4);
END_IF
                      
END_ACTION

ACTION TEST_CASE_1_EXEC:
                        IF vTestCases[0].state = utTestCaseStates.RUNNING THEN
	(*Run the test case*)
	IF assertGreater_LDATE(vTestCase1_act, vTestCase1_xp) THEN
		vTestCases[0].state := utTestCaseStates.PASSED;
		vTestCases[0].msg := 'Parameter act was greater than xp and function returned TRUE -> PASS';
	ELSE
		vTestCases[0].state := utTestCaseStates.FAILED;
		vTestCases[0].msg := 'Parameter act was greater than xp and function returned FALSE -> FAIL';
	END_IF
END_IF
                      
END_ACTION

ACTION TEST_CASE_2_SETUP:
                        IF vTestCases[1].state = utTestCaseStates.SETUP THEN
	(*Setup the test case information*)
	vTestCases[1].id := 2;
    vTestCases[1].desc[0] := 'RETURNS FALSE WHEN PARAMETER ACT LESS THAN XP';
    vTestCases[1].desc[1] := 'Tests if the function returns False if the parameter act is less than parameter xp';
	vTestCases[1].desc[2] := 'PASS IF: Return value is FALSE';
	
	(*Setup needed variables*)
	vTestCase2_act := REAL_TO_LDATE(8.4);
	vTestCase2_xp := REAL_TO_LDATE(85.4);
END_IF
                      
END_ACTION

ACTION TEST_CASE_2_EXEC:
                        IF vTestCases[1].state = utTestCaseStates.RUNNING THEN
	(*Run the test case*)
	IF NOT assertGreater_LDATE(vTestCase2_act, vTestCase2_xp) THEN
		vTestCases[1].state := utTestCaseStates.PASSED;
		vTestCases[1].msg := 'Parameter act was less than xp and function returned FALSE -> PASS';
	ELSE
		vTestCases[1].state := utTestCaseStates.FAILED;
		vTestCases[1].msg := 'Parameter act was less than xp and function returned TRUE -> FAIL';
	END_IF
END_IF
                      
END_ACTION
END_PROGRAM

PROGRAM test_assertGreaterEqual_UDINT
  VAR
    vTestCases : ARRAY[0..20] OF utTestCase;  (* Definition of all test cases for this POU *)
    testRunner : utTestSuite;  (* Test Suite fb instance to run the tests *)
    vRunAll : BOOL;  (* Manual command to run all tests for this POU *)
    vResetAll : BOOL;  (* Manual command to reset all tests for this POU *)
    vTestCase1_act : UDINT;  (* Test data 1 of test case 1 *)
    vTestCase1_xp : UDINT;  (* Test data 2 of test case 1 *)
    vTestCase2_act : UDINT;  (* Test data 1 of test case 2 *)
    vTestCase2_xp : UDINT;  (* Test data 2 of test case 2 *)
    vTestCase3_act : UDINT;  (* Test data 1 of test case 3 *)
    vTestCase3_xp : UDINT;  (* Test data 2 of test case 3 *)
  END_VAR

                    (*Run the test cases*)
TEST_CASE_1_SETUP();
TEST_CASE_1_EXEC();

TEST_CASE_2_SETUP();
TEST_CASE_2_EXEC();

TEST_CASE_3_SETUP();
TEST_CASE_3_EXEC();

(*Instantiate the test runner*)
testRunner(
	Id := 81,
	Name := 'assertGreaterEqual_UDINT',
    RunTests := GVL.RunAll OR vRunAll,
	ResetTests := GVL.ResetAll OR vResetAll,
	TestCases:=vTestCases);

(*Report the results to the collection global*)
GVL.Results[testRunner.Id] := testRunner.Summary;
                  

ACTION TEST_CASE_1_SETUP:
                        IF vTestCases[0].state = utTestCaseStates.SETUP THEN
	(*Setup the test case information*)
	vTestCases[0].id := 1;
	vTestCases[0].desc[0] := 'RETURNS TRUE WHEN PARAMETER ACT GREATER THAN XP';
    vTestCases[0].desc[1] := 'Tests if the function returns True if the parameter act is greater than parameter xp';
	vTestCases[0].desc[2] := 'PASS IF: Return value is TRUE';
	
	(*Setup needed variables*)
	vTestCase1_act := REAL_TO_UDINT(115.4);
	vTestCase1_xp := REAL_TO_UDINT(85.4);
END_IF
                      
END_ACTION

ACTION TEST_CASE_1_EXEC:
                        IF vTestCases[0].state = utTestCaseStates.RUNNING THEN
	(*Run the test case*)
	IF assertGreaterEqual_UDINT(vTestCase1_act, vTestCase1_xp) THEN
		vTestCases[0].state := utTestCaseStates.PASSED;
		vTestCases[0].msg := 'Parameter act was greater than xp and function returned TRUE -> PASS';
	ELSE
		vTestCases[0].state := utTestCaseStates.FAILED;
		vTestCases[0].msg := 'Parameter act was greater than xp and function returned FALSE -> FAIL';
	END_IF
END_IF
                      
END_ACTION

ACTION TEST_CASE_2_SETUP:
                        IF vTestCases[1].state = utTestCaseStates.SETUP THEN
	(*Setup the test case information*)
	vTestCases[1].id := 2;
    vTestCases[1].desc[0] := 'RETURNS TRUE WHEN PARAMETER ACT EQUAL TO XP';
    vTestCases[1].desc[1] := 'Tests if the function returns True if the parameter act is equal to parameter xp';
	vTestCases[1].desc[2] := 'PASS IF: Return value is TRUE';
	
	(*Setup needed variables*)
	vTestCase2_act := REAL_TO_UDINT(115.4);
	vTestCase2_xp := REAL_TO_UDINT(115.4);
END_IF
                      
END_ACTION

ACTION TEST_CASE_2_EXEC:
                        IF vTestCases[1].state = utTestCaseStates.RUNNING THEN
	(*Run the test case*)
	IF assertGreaterEqual_UDINT(vTestCase2_act, vTestCase2_xp) THEN
		vTestCases[1].state := utTestCaseStates.PASSED;
		vTestCases[1].msg := 'Parameter act was equal to xp and function returned TRUE -> PASS';
	ELSE
		vTestCases[1].state := utTestCaseStates.FAILED;
		vTestCases[1].msg := 'Parameter act was equal to xp and function returned FALSE -> FAIL';
	END_IF
END_IF
                      
END_ACTION

ACTION TEST_CASE_3_SETUP:
                        IF vTestCases[2].state = utTestCaseStates.SETUP THEN
	(*Setup the test case information*)
	vTestCases[2].id := 3;
    vTestCases[2].desc[0] := 'RETURNS FALSE WHEN PARAMETER ACT LESS THAN XP';
    vTestCases[2].desc[1] := 'Tests if the function returns False if the parameter act is less than parameter xp';
	vTestCases[2].desc[2] := 'PASS IF: Return value is FALSE';
	
	(*Setup needed variables*)
	vTestCase3_act := REAL_TO_UDINT(85.4);
	vTestCase3_xp := REAL_TO_UDINT(115.4);
END_IF
                      
END_ACTION

ACTION TEST_CASE_3_EXEC:
                        IF vTestCases[2].state = utTestCaseStates.RUNNING THEN
	(*Run the test case*)
	IF NOT assertGreaterEqual_UDINT(vTestCase3_act, vTestCase3_xp) THEN
		vTestCases[2].state := utTestCaseStates.PASSED;
		vTestCases[2].msg := 'Parameter act was less than xp and function returned FALSE -> PASS';
	ELSE
		vTestCases[2].state := utTestCaseStates.FAILED;
		vTestCases[2].msg := 'Parameter act was less than xp and function returned TRUE -> FAIL';
	END_IF
END_IF
                      
END_ACTION
END_PROGRAM

PROGRAM test_assertGreaterEqual_DATE
  VAR
    vTestCases : ARRAY[0..20] OF utTestCase;  (* Definition of all test cases for this POU *)
    testRunner : utTestSuite;  (* Test Suite fb instance to run the tests *)
    vRunAll : BOOL;  (* Manual command to run all tests for this POU *)
    vResetAll : BOOL;  (* Manual command to reset all tests for this POU *)
    vTestCase1_act : DATE;  (* Test data 1 of test case 1 *)
    vTestCase1_xp : DATE;  (* Test data 2 of test case 1 *)
    vTestCase2_act : DATE;  (* Test data 1 of test case 2 *)
    vTestCase2_xp : DATE;  (* Test data 2 of test case 2 *)
    vTestCase3_act : DATE;  (* Test data 1 of test case 3 *)
    vTestCase3_xp : DATE;  (* Test data 2 of test case 3 *)
  END_VAR

                    (*Run the test cases*)
TEST_CASE_1_SETUP();
TEST_CASE_1_EXEC();

TEST_CASE_2_SETUP();
TEST_CASE_2_EXEC();

TEST_CASE_3_SETUP();
TEST_CASE_3_EXEC();

(*Instantiate the test runner*)
testRunner(
	Id := 88,
	Name := 'assertGreaterEqual_DATE',
    RunTests := GVL.RunAll OR vRunAll,
	ResetTests := GVL.ResetAll OR vResetAll,
	TestCases:=vTestCases);

(*Report the results to the collection global*)
GVL.Results[testRunner.Id] := testRunner.Summary;
                  

ACTION TEST_CASE_1_SETUP:
                        IF vTestCases[0].state = utTestCaseStates.SETUP THEN
	(*Setup the test case information*)
	vTestCases[0].id := 1;
	vTestCases[0].desc[0] := 'RETURNS TRUE WHEN PARAMETER ACT GREATER THAN XP';
    vTestCases[0].desc[1] := 'Tests if the function returns True if the parameter act is greater than parameter xp';
	vTestCases[0].desc[2] := 'PASS IF: Return value is TRUE';
	
	(*Setup needed variables*)
	vTestCase1_act := REAL_TO_DATE(115.4);
	vTestCase1_xp := REAL_TO_DATE(85.4);
END_IF
                      
END_ACTION

ACTION TEST_CASE_1_EXEC:
                        IF vTestCases[0].state = utTestCaseStates.RUNNING THEN
	(*Run the test case*)
	IF assertGreaterEqual_DATE(vTestCase1_act, vTestCase1_xp) THEN
		vTestCases[0].state := utTestCaseStates.PASSED;
		vTestCases[0].msg := 'Parameter act was greater than xp and function returned TRUE -> PASS';
	ELSE
		vTestCases[0].state := utTestCaseStates.FAILED;
		vTestCases[0].msg := 'Parameter act was greater than xp and function returned FALSE -> FAIL';
	END_IF
END_IF
                      
END_ACTION

ACTION TEST_CASE_2_SETUP:
                        IF vTestCases[1].state = utTestCaseStates.SETUP THEN
	(*Setup the test case information*)
	vTestCases[1].id := 2;
    vTestCases[1].desc[0] := 'RETURNS TRUE WHEN PARAMETER ACT EQUAL TO XP';
    vTestCases[1].desc[1] := 'Tests if the function returns True if the parameter act is equal to parameter xp';
	vTestCases[1].desc[2] := 'PASS IF: Return value is TRUE';
	
